# B&R Automation Studio project x20ost (part 6)

#### bnrmessage.h
```c
/********************************************************************
 * COPYRIGHT -- Kontora
 ********************************************************************
 * Program: bnrmain
 * File: bnraninput.h
 * Author: Abramenya
 * Created: January 19, 2009
 *******************************************************************/

#ifndef __MESSAGE_H__
#define __MESSAGE_H__
#include "typedefs.h"
typedef void (*CCPFN)(void);
//Message For My System
#ifdef WIN32
typedef struct _tagCANnode_typ
{
	BOOL enable;
	UINT node_nr;
	UINT status;
}CANnode_typ;

typedef struct _tagCANopen_typ
{
	BOOL enable;
	UINT baud_rate;
	UINT cob_anz;
	UINT device;
}CANopen_typ;

typedef struct _tagFRM_xopen_typ
{
	BOOL   enable;
	UDINT	device;
	UDINT	mode;
	UDINT	config;
	UINT	status;
	UDINT	*ident;
	BYTE	internal[27];
}FRM_xopen_typ;
typedef struct _tagFRM_close_typ
{
	BOOL   enable;
	UDINT  *ident;
	UINT   status;
	BYTE   internal[27];
}FRM_close_typ;
typedef struct _tagXOPENCONFIG
{
	UINT   idle;
	UINT   delimc;
	USINT  delim[2];
	UINT   tx_cnt;
	UINT   rx_cnt;
	UINT   tx_len;
	UINT   rx_len;
	UINT   argc;
	UDINT  *argv;
}XOPENCONFIG;
typedef struct _tagFRM_gbuf_typ
{
	BOOL   enable;
	UDINT  *ident;
	UINT   status;
	UDINT  *buffer;
	UINT	buflng;
	BYTE	internal[27];
}FRM_gbuf_typ;
//Client
typedef struct _tagFRM_rbuf_typ
{
	BOOL   enable;
	UDINT	*ident;
	UDINT	*buffer;
	UINT	buflng;
	UINT	status;
	BYTE	internal[27];
}FRM_rbuf_typ;
typedef struct _tagFRM_robuf_typ
{
	BOOL   enable;
	UDINT	*ident;
	UDINT	*buffer;
	UINT	buflng;
	UINT	status;
	BYTE	internal[27];
}FRM_robuf_typ;
typedef struct _tagFRM_write_typ
{
	BOOL   enable;
	UDINT  *ident;
	UDINT  *buffer;
	UINT   buflng;
	UINT   status;
	BYTE   internal[27];

}FRM_write_typ;
typedef struct _tagFRM_read_typ
{
	BOOL   enable;
	UDINT  *ident;
	UINT   status;
	UDINT  *buffer;
	UINT   buflng;
	BYTE   internal[27];
}FRM_read_typ;
typedef struct _tagSysInfo
{
    BYTE byInfo;
}SYSxinfo_typ;
typedef struct _tagRTCtime_typ
{
    WORD year;
    BYTE month;
    BYTE day;
    BYTE hour;
    BYTE minute;
    BYTE second;
    WORD millisec;
}RTCtime_typ;
int SYSxinfo(SYSxinfo_typ*);
#endif
typedef struct _tagGetParam
{
    WORD wParam0;
	WORD wParam1;
	WORD wParam2;
	WORD wParam3;
}SGETPARAM;
typedef struct _msgPLCCommand
{
    WORD m_swLen;
	BYTE m_sbyFor;
	BYTE m_sbyType;
    BYTE m_sbyDevID;
	BYTE m_sbyInfo[70];
}SPLCCOMM;
typedef struct _msgSystem0
{
    WORD m_swLen;
    BYTE m_sbyFrom;
	BYTE m_sbyFor;
	BYTE m_sbyIntType;
	BYTE m_sbyServerID;
	BYTE m_sbyType;
    BYTE m_sbyDirection;
    BYTE m_sbySensor;
	BYTE m_sbyInfo[350];
}SMESSAGE;
typedef struct _msgSystem00
{
    WORD m_swLen;
    BYTE m_sbyFrom;
	BYTE m_sbyFor;
	BYTE m_sbyIntType;
	BYTE m_sbyServerID;
	BYTE m_sbyType;
    BYTE m_sbyDirection;
    BYTE m_sbySensor;
	BYTE m_sbyInfo[2000];
}SLMESSAGE;
typedef struct _msgShSystem0
{
    WORD m_swLen;
    BYTE m_sbyFrom;
	BYTE m_sbyFor;
	BYTE m_sbyIntType;
	BYTE m_sbyServerID;
	BYTE m_sbyType;
    BYTE m_sbyDirection;
    BYTE m_sbySensor;
	BYTE m_sbyInfo[200];
}SHMESSAGE;
typedef struct _msgShSystem1
{
    WORD m_swLen;
    BYTE m_sbyFrom;
	BYTE m_sbyFor;
	BYTE m_sbyIntType;
	BYTE m_sbyServerID;
	BYTE m_sbyType;
    BYTE m_sbyDirection;
    BYTE m_sbySensor;
	BYTE m_sbyInfo[30];
}SHORTMESSAGE;
typedef struct _tagJob
{
	CCPFN pfnProcAddres;
	BYTE  byPeriod;
	BYTE  byStateProc;
	SINT  chProcName[50];
}SJOBINFO;

typedef struct _tagTcpAddres
{
    BYTE byAddr0;
	BYTE byAddr1;
	BYTE byAddr2;
	BYTE byAddr3;
}STCPADDR;
typedef struct _tagArmInterface
{
	BYTE byNumber;
    BYTE byType;
	BYTE byPortRate;
	BYTE byAmTCPPort;
	DWORD dwpPortNumber[DEV_MAX_TCP_PORT];
	STCPADDR stTcpAddr;
	SINT chTcpAddr[30];
}SARMINTERFACE;
typedef struct _tagHardPinConfig
{
	BYTE byPinNumber;
	BYTE byPinType;
	BYTE byPinState;
	PVOID pvValue;
}SHARDPIN;
typedef struct _tagHardSlotConfig
{
	BYTE bySlotNumber;
	BYTE bySlotType;
	BYTE byPinAmout;
	BYTE byState;
	BYTE byAlmState;
	PVOID pvAlmState;
	PVOID *pvAlmPin;
	PVOID *pvPin;
}SHARDSLOT;
typedef struct _tagKpParam
{
    BYTE byKpID;
	BYTE byStoreMode;
	BYTE byAmCall;
	BYTE byCallPeriod;
	//BYTE bySetChann;
	SINT byPassword[20];
	SINT byPhone0[20];
	SINT byPhone1[20];
	SINT byPhone2[20];
}SKPPARAM;
typedef struct _tagHardComputer
{
    BYTE byComputerType;
	BYTE bySystemID;
    SINT chComputerName[DEV_MAX_TEXT_NAME];
	SINT chProgrammVersion[DEV_MAX_TEXT_NAME];
    SINT chDateOfWrite[DEV_MAX_TEXT_NAME];
	BYTE bySlotAmout;
	BYTE byArmAmout;
	SKPPARAM *pKpParam;
	SARMINTERFACE *pArmInterface[DEV_MAX_ARM_PORT];
	SHARDSLOT sSlot[DEV_MAX_SLOTS_PS260];
}SHARDCOMPUTERTABLE;
typedef struct _tagSensorInitTable
{
    INT  iLoLimitValue;
	INT  iHiLimitValue;
}SENSORINITTABLE;
/*
pT->m_sSNSParam.dY_max    = 20.0;
pT->m_sSNSParam.Kp        = 0.4;
pT->m_sSNSParam.Tn        = 6000.0;
pT->m_sSNSParam.Tv        = 0.0;
pT->m_sSNSParam.Tf        = 1.0;
pT->m_sSNSParam.Kw        = 1.0;
pT->m_sSNSParam.Kfbk      = 1.0;
pT->m_sLCPid.A            = 0;//500;
pT->m_sLCPid.Y_man	      = 0;
*/
typedef struct _tagSensorParamTable
{
    REAL m_swResistance;
    REAL m_swHiLimit;
    REAL m_swLoLimit;
    REAL m_swHiAlLimit;
    REAL m_swLoAlLimit;
    REAL m_swHiOper;
    REAL m_swLoOper;
    REAL m_swInitValue;
	REAL m_rlDy;
	REAL m_rlKp;
	REAL m_rlTn;
	REAL m_rlKw;
	REAL m_rlKfbk;
	REAL m_rlTv;
	REAL m_rlTf;
	INT16 m_rlA;
	INT16 m_rlYman;
	BYTE m_byFilterOn;
	BYTE m_swPidDiffMode;
	WORD m_swMaxAcpInp;
	WORD m_swMaxAcpOut;
	BYTE m_byID;
    BYTE bySrcSlotNumber;
	BYTE bySrcPinNumber;
    BYTE m_snType;
    BYTE m_sbyParamType;
    BYTE m_sbyInpState;
    BYTE m_sbyOutState;
    BYTE m_sbyMode;
	BYTE m_sbyPmode;
	BYTE m_sbyOmode;
	REAL m_srOmin;
	REAL m_srOmax;
	WORD m_swOpenTime;
	SINT m_chSNname[10];
}SNSPARAMTABLE;

typedef struct _tagOutGate
{
	WORD wLoLimit;
	WORD wHiLimit;
	WORD wCurrOpen;
	WORD wOpenTime;
	REAL rMinRamp;
	REAL rMaxRamp;
	BYTE byOType;
	BYTE byMode;
	BYTE byID;
	BYTE byType;
    BYTE byOutSlotNumber;
	BYTE byOutPinNumber;
	SINT chName[10];
}SOUTGATE;
typedef struct _tagSensorInputGates
{
  BYTE byAmInGate;
  SNSPARAMTABLE mIn[12];
}SINPUTGATE;
typedef struct _tagSensorOutputGates
{
	BYTE byAmOutGate;
	SOUTGATE mOut[12];
}SOUTPUTGATE;
typedef struct _tagPinGate
{
	BYTE sbySlot;
	BYTE sbyPin;
}SPINGATE;
typedef struct _tagDigitalGate
{
    WORD swAmpin;
	SPINGATE sPinGate[32];
}SDIGGATE;
typedef struct _tagDigitalGates
{
    BYTE byAmGate;
	SDIGGATE sIoGate[10];
}SDIGGATES;
typedef struct _tagSwitchingTable
{
    #if MYSYSTEM_ID != 5
	 BYTE bySensorID;
	 PVOID sSensorParamTable;
	 TStateList *m_pStateList;
	 BYTE bySwitchCommand;
	 BOOL blEnable;
	 BYTE byAmOutGate;
	 PVOID sOutGate[DEV_AMT_GATE_SNS];
	#else
	 BYTE bySensorID;
     BYTE bySlot;
	 BYTE byPin;
	 BYTE byType;
    #endif
}SSWITCHTABLE;
typedef struct _tagDirectionTable
{
    BYTE byDirectionID;
	BYTE byDirectionCode;
	BYTE byAmSwitching;
	BYTE byAmTI;
	BYTE byAmTS;
	BYTE byAmTU;
	BYTE byAmTR;

	PVOID pvIn;
	PVOID pvOut;
	PVOID pSwitchTable[DEV_AMT_SWC_IDIR];
}SDIRTABLE;
typedef struct _tagSoftSwitchingConfig
{
	BYTE byTableVersion;
	SINT chTableVersionName[DEV_MAX_TEXT_NAME];
	BYTE byAmDirection;
	SDIRTABLE sDirectionTable[DEV_AMT_DIR_INST];
}SSOFTSWITCHTABLE;
//Kp Tag
typedef struct _tagTime
{
    BYTE tDay;
	BYTE tMonth;
	BYTE tYear;
	BYTE tHour;
	BYTE tMin;
	BYTE tSec;
	BYTE tMSecL;
	BYTE tMSecH;
}STIME;
typedef struct _tagKpEvent
{
	WORD wLen;
	BYTE byType;
    BYTE byAddr;
	BYTE byCause;
    WORD wValue;
    STIME sTime;
}SKPEVENT;
typedef struct _tagQueryReqAddr
{
	WORD wSize;
	BYTE byA0;
	BYTE byA1;
	BYTE byA2;
}SREGADDR;
typedef struct _tagReqParam
{
	WORD wSize;
	WORD wParam;
	BYTE byA0;
	BYTE byA1;
	BYTE byA2;
}SREGPARAM;
//Датчик температуры
typedef struct _tagTTMData
{
	WORD wJob;
	WORD wParam;
}STTMDATA;
/*
typedef struct _tagTTMDatas
{
	BYTE Count;
	BYTE byType;
	STTMDATA sDT[2];
}STTMDATAS;
*/
typedef struct _tagTTMParam
{
	BYTE byID;
	BYTE byAmParam;
	BYTE byType;
	BYTE bySlot;
	BYTE byPin;
	BYTE byAlmState;
	BYTE byState;
	STTMDATA sDT;
}STTMPARAM;
typedef struct _tagTTMParams
{
	BYTE byAmSlot;
	BYTE byType;
	STTMPARAM sTTM[4];
}STTMPARAMS;
//Датчик давления
typedef struct _tagTPRData
{
	WORD wJob;
	WORD wParam;
}SPRMDATA;
/*
typedef struct _tagTPRDatas
{
	BYTE Count;
	BYTE byType;
	SPRMDATA sDT[2];
}SPRMDATAS;
*/
typedef struct _tagTPRParam
{
	BYTE byID;
	BYTE byAmParam;
	BYTE byType;
	BYTE bySlot;
	BYTE byPin;
	BYTE byAlmState;
	BYTE byState;
	SPRMDATA sDT;
}STPRPARAM;
typedef struct _tagTPRParams
{
	BYTE byAmSlot;
	BYTE byType;
	STPRPARAM sTPR[4];
}STPRPARAMS;
//Счетчики
typedef struct _tagTCData
{
	REAL fKoeff;
	DWORD dwParam;
}STCDATA;
/*
typedef struct _tagTCDatas
{
	BYTE Count;
	BYTE byType;
	STCDATA sDT[16];
}STCDATAS;
*/
typedef struct _tagTCParam
{
	BYTE byID;
	BYTE byAmParam;
	BYTE byType;
	BYTE bySlot;
	BYTE byPin;
	BYTE byAlmState;
	BYTE byState;
	DWORD dwMaxFreq;
	STCDATA sDT;
}STCPARAM;
typedef struct _tagTCParams
{
	BYTE byAmSlot;
	BYTE byType;
	STCPARAM sTC[18];
}STCPARAMS;
//Управляемые краны
typedef struct _tagTKData
{
	BYTE byStOP;
	BYTE byStCL;
	BYTE byStMD;
    WORD wMaxOpenTime;
    REAL fJobOpen;
    REAL fOpenState;
}STKDATA;
/*
typedef struct _tagTKDatas
{
	BYTE Count;
	BYTE byType;
	STKDATA sDT[4];
}STKDATAS;
*/
typedef struct _tagTKParam
{
	BYTE byID;
	BYTE byAmParam;
	BYTE byType;
	BYTE bySlot;
	BYTE byPin;
	BYTE bySlot1;
	BYTE byPin1;
    STKDATA sDT;
}STKPARAM;
typedef struct _tagTKParams
{
	BYTE byAmSlot;
	BYTE byType;
	STKPARAM sTK[5];
}STKPARAMS;
//Измеритель уровня
typedef struct _tagLVData
{
	WORD wSt0;
	WORD wJob0;
	WORD wJob1;
	WORD wParam;
}SLVDATA;
/*
typedef struct _tagPUDatas
{
	BYTE Count;
	BYTE byType;
	SPUDATA sDT[2];
}SPUDATAS;
*/
typedef struct _tagLVParam
{
	BYTE byID;
	BYTE byAmParam;
	BYTE byType;
	BYTE bySlot;
	BYTE byPin;
	BYTE bySlot1;
	BYTE byPin1;
    SLVDATA sDT;
}SLVPARAM;
typedef struct _tagLVParams
{
	BYTE byAmSlot;
	BYTE byType;
	SLVPARAM sLV[2];
}SLVPARAMS;
//Переключатель режима
typedef struct _tagPLData
{
	BYTE byParam;
}SPLDATA;
typedef struct _tagPLParam
{
	BYTE byID;
	BYTE byAmParam;
	BYTE byType;
	BYTE bySlot;
	BYTE byPin;
    SPLDATA sDT;
}SPLPARAM;
typedef struct _tagPLParams
{
	BYTE byAmSlot;
	BYTE byType;
	SPLPARAM sPL[2];
}SPLPARAMS;
//Таймер операции
typedef struct _tagTMData
{
	WORD wJob;
	WORD wParam;
}STMDATA;
typedef struct _tagTMParam
{
	BYTE byID;
	BYTE byAmParam;
	BYTE byType;
	BYTE bySlot;
	BYTE byPin;
    STMDATA sDT;
}STMPARAM;
typedef struct _tagTMParams
{
	BYTE byAmSlot;
	BYTE byType;
	STMPARAM sTM[2];
}STMPARAMS;
//Перекидное устройство
typedef struct _tagPUData
{
	WORD wSt0;
	WORD dwTimeConst;
	WORD dwOpenTime;
}SPUDATA;
/*
typedef struct _tagPUDatas
{
	BYTE Count;
	BYTE byType;
	SPUDATA sDT[2];
}SPUDATAS;
*/
typedef struct _tagPUParam
{
	BYTE byID;
	BYTE byAmParam;
	BYTE byType;
	BYTE bySlot;
	BYTE byPin;
	BYTE bySlot1;
	BYTE byPin1;
	BYTE bySlot2;
	BYTE byPin2;
	BYTE bySlot3;
	BYTE byPin3;
    SPUDATA sDT;
}SPUPARAM;
typedef struct _tagPUParams
{
	BYTE byAmSlot;
	BYTE byType;
	SPUPARAM sTPU[2];
}SPUPARAMS;
//Частотный привод
typedef struct _tagTFData
{
	//BYTE byStartST;
	//BYTE byStopST;
	//BYTE byAlST0;
	//BYTE byAlST1;
    WORD wSt0;
	WORD wTask;
	WORD wParam;
}STFDATA;
/*
typedef struct _tagTFDatas
{
	BYTE Count;
	BYTE byType;
	STFDATA sDT[3];
}STFDATAS;
*/
typedef struct _tagTFParam
{
	BYTE byID;
	BYTE byAmParam;
	BYTE byType;
	BYTE bySlot; //Для задания
	BYTE byPin;  //Для задания

	BYTE bySlot1; //Запуск
	BYTE byPin1;  //Запуск

	BYTE bySlot2; //Останов
	BYTE byPin2;  //Останов

	BYTE bySlot3; //Авария1
	BYTE byPin3;  //Авария1

	BYTE bySlot4; //Авария2
	BYTE byPin4;  //Авария2
    STFDATA sDT;
}STFPARAM;
typedef struct _tagTFParams
{
	BYTE byAmSlot;
	BYTE byType;
	STFPARAM sTF[4];
}STFPARAMS;
//Телеиндикация
typedef struct _tagTIParam
{
	BYTE byID;
	BYTE byAmParam;
	BYTE byType;
	BYTE bySlot;
	BYTE byPin;
	BYTE byAlmState;
	BYTE byState;
	BYTE byPriority;
	BYTE byDrTimer;
	WORD wHiLimit;
	WORD wHiGister;
	WORD wLoGister;
	WORD wLoLimit;
	WORD wLo;
	WORD wHi;
	WORD wEvPercent;
	WORD wParam;
}STIPARAM;
typedef struct _tagTIParams
{
	BYTE byAmSlot;
	BYTE byType;
	STIPARAM sTI[32];
}STIPARAMS;

//Весы
typedef struct _tagTVSData
{
	BYTE byData[11];
}STVSDATA;
typedef struct _tagTVSParam
{
	BYTE byID;
	BYTE byAmParam;
	BYTE byType;
	STVSDATA sDT;
}STVSPARAM;
typedef struct _tagTVSarams
{
	BYTE byAmSlot;
	BYTE byType;
	STIPARAM sTVS[2];
}STVSPARAMS;
//Телесигнализация(дискретное)
typedef struct _tagTSParam
{
	BYTE byID;
	BYTE byAmParam;
	BYTE byType;
	BYTE bySlot;
	BYTE byPin;
	BYTE byAlmState;
	BYTE byState;
	BYTE byPriority;
	BYTE byCRemPulce;
    BYTE byCSetPulce;
	BYTE byAlarmMode;
    BYTE byParam;
}STSPARAM;
typedef struct _tagTSParams
{
	BYTE byAmSlot;
	BYTE byType;
	STSPARAM sTS[20];
}STSPARAMS;

//Телесигнализация1(дискретное)
typedef struct _tagTSMData
{
	BYTE byParam;
}STSMDATA;
/*
typedef struct _tagTSMDatas
{
	BYTE Count;
	BYTE byType;
	STSMDATA sDT[19];
}STSMDATAS;
*/
typedef struct _tagTSMParam
{
	BYTE byID;
	BYTE byAmParam;
	BYTE byType;
	BYTE bySlot;
	BYTE byPin;
	BYTE byAlmState;
	BYTE byState;
	BYTE byPriority;
	BYTE byCRemPulce;
    BYTE byCSetPulce;
	BYTE byAlarmMode;
    STSMDATA sDT;
}STSMPARAM;
typedef struct _tagTSMParams
{
	BYTE byAmSlot;
	BYTE byType;
	STSPARAM sTS[20];
}STSMPARAMS;

//Аварии
typedef struct _tagTALData
{
	WORD wParam;
}STALDATA;
typedef struct _tagTALaram
{
	BYTE byID;
	BYTE byAmParam;
	BYTE byType;
	BYTE bySlot;
	BYTE byPin;
	BYTE byAlmState;
	BYTE byState;
    STALDATA sDT;
}STALPARAM;
typedef struct _tagTALParams
{
	BYTE byAmSlot;
	BYTE byType;
	STALPARAM sTA[2];
}STALPARAMS;

//Телеуправление(дискретное)
typedef struct _tagTUParam
{
	BYTE byID;
	BYTE byAmParam;
	BYTE byType;
	BYTE bySlot;
	BYTE byPin;
	BYTE byAlmState;
	BYTE byState;
	BYTE byPulceType;
    BYTE byCSetPulce;
	BYTE byParam;
}STUPARAM;
typedef struct _tagTUParams
{
	BYTE byAmSlot;
	BYTE byType;
	STUPARAM sTU[64];
}STUPARAMS;

//Телеуправление1(дискретное)
typedef struct _tagTUMData
{
	BYTE byParam;
}STUMDATA;
typedef struct _tagTUMParam
{
	BYTE byID;
	BYTE byAmParam;
	BYTE byType;
	BYTE bySlot;
	BYTE byPin;
	BYTE byAlmState;
	BYTE byState;
	BYTE byPulceType;
    DWORD byCSetPulce;
	STUMDATA sDT;
}STUMPARAM;
typedef struct _tagTUMParams
{
	BYTE byAmSlot;
	BYTE byType;
	STUMPARAM sTU[16];
}STUMPARAMS;

//Модуль слежения
typedef struct _tagODSData
{
	//BYTE byAutoStart;
	//BYTE byPreStart;
	//BYTE byStart;
	//BYTE byStop;
	//BYTE byFinish;
    //BYTE byMode;
    DWORD wSt0;
	WORD wJTMPreStart;
	WORD wTMPreStart;
	WORD wJTMStart;
	WORD wTMStart;
	WORD wJTMWait;
	WORD wTMWait;
}SOBSMDATA;
typedef struct _tagOBSParam
{
	BYTE byID;
	BYTE byAmParam;
	BYTE byType;
	BYTE bySlot;
	BYTE byPin;
	BYTE byAlmState;
	BYTE byState;
	SOBSMDATA sDT;
}SOBSPARAM;
typedef struct _tagOBSParams
{
	BYTE byAmSlot;
	BYTE byType;
	SOBSPARAM sOS[1];
}SOBSPARAMS;

/*
&nTPR,
&nTTM,
&nTC,
&nTF,
&nTKP,
&nTPU,
&nTS,
&nTU,
*/
typedef struct _tagObserveTable
{
    SPRMDATA nTPR[2];
    STTMDATA nTTM[2];
	STCDATA  nTC[16];
	STFDATA  nTF[3];
	STKDATA  nTKP[4];
	SPUDATA  nPU[2];
	STSMDATA nTS[15];
	STUMDATA nTU[10];
	STVSDATA nTVS[2];
	SLVDATA  nLV[1];
	SPLDATA  nPL[1];
	STMDATA  nTM[1];
	STALDATA nTAL[2];
}STOUTTBL;
typedef struct _tagCDataCommand
{
     WORD wDeviceID;
     BYTE byParam0;
     BYTE byParam1;
     BYTE byParam2;
     WORD wParam0;
     WORD wParam1;
     WORD wParam2;
     REAL fParam0;
     REAL fParam1;
     REAL fParam2;
}CDataCommand;
typedef struct _tagContenstTable
{
	BYTE byKpID;
	BYTE byDefSett;
	//#if (MYSYSTEM_ID == 0)||(MYSYSTEM_ID == 1)||(MYSYSTEM_ID == 2)||(MYSYSTEM_ID == 3)
	//REAL mInResistance[16];
    //SINPUTGATE  sInGate;
    ///SOUTPUTGATE sOutGate;
	//WORD m_wLayerMode;
    //#elif MYSYSTEM_ID == 4
	//DWORD m_dwOutState[32];
    //#elif MYSYSTEM_ID == 5
	SKPPARAM  sKP;
	SARMINTERFACE sARM;
	STIPARAMS sTI;
	STSPARAMS sTS;
	STUPARAMS sTU;
    //#endif
}SCONTENSTTABLE;
#endif
```

#### bnrmodule101.h
```c
/********************************************************************
 * COPYRIGHT -- Kontora
 ********************************************************************
 * Program: bnrmain
 * File: bnraninput.h
 * Author: Abramenya
 * Created: January 19, 2009
 *******************************************************************/

#ifndef __MODULE101_H__
#define __MODULE101_H__
#include "typedefs.h"
#include "bnrcyclicsystem.h"
#include "bnrregedit.h"
Class CModule101
{
	 void (*CCModule101)(This);
	 void (*DCModule101)(This);
Public
     void (*Init)(This);
     BOOL (*LoLevelHandler)(This,SMESSAGE *pMsg);
     BOOL (*HiLevelHandler)(This,SMESSAGE *pMsg);
	 BOOL (*SendMessage)(This,BYTE,BYTE);
	 BYTE (*CreateCRC)(This,BYTE *pMsg,BYTE byLen);
	 BYTE (*AddADSU)(This,BYTE *pMsg,BYTE byNum);
	 BYTE (*AddADSU1)(This,BYTE *pMsg,BYTE byNum);
	 BYTE (*PackADSU)(This,BYTE *pMsg);
	 WORD (*GetW)(This,BYTE *pbyParam);
	 BOOL (*GetSettings)(This);
	 BOOL (*SetSettings)(This);
	 void (*CopyW)(This,PVOID pvDst,PVOID pvSrc);
	 BOOL (*SendBroadcast)(This,SMESSAGE *pMsg);
	 BYTE (*AddBroadADSU)(This,BYTE *pMsg,SKPEVENT *pEV);
	 BOOL (*Autorisation)(This,WORD wKeyCode,BYTE byKpID);
     Virtual BOOL (*HandleTask)(This,TTask* pvTask);
     Virtual BOOL (*EventHandler)(This,SMESSAGE *pMsg);
	 Virtual TStateList* (*GetStateList)(This);
     //Virtual void (*CyclicProc)(This);
	 DECLARE_IMPLEMENT_BASE(CCyclicSystem)
Private
     CRegModule m_nRM;
     BYTE m_byModuleID;
	 BOOL m_blRepFree;
	 //STISTAG  m_sTiTsMsg;
	 SREGADDR m_pA;
	 SREGPARAM m_nRD;
	 SMESSAGE *m_pOutMsg;
	 SMESSAGE m_sOutMsg;
	 SMESSAGE m_sSvOutMsg;
}
DECLARE_DEFINITION(CModule101)
#define TIMER_SRR_00 10

/*
typedef struct   {
BYTE bt0; // аҐ§Ґаў ў ­ з «Ґ
BYTE bt1; //
BYTE Len;
unsigned nGlUnit:6; //ЙНННН»
unsigned nLocUnit:5;//є    є
unsigned nP1:4;      //є ID є
unsigned bit1:1;
unsigned nP2:11;
unsigned nP3:5;
BYTE Data[0x100-7];
} MSG_FPO1;
*/
typedef struct _tagAdsuHead
{
    BYTE Type;
    BYTE VSQ;
    BYTE Cause;
    //BYTE Ordinator;
    BYTE CAA00;
    BYTE CAA01;
}SADSUHEAD;
typedef struct _tagIEA
{
    BYTE IOA00;
    BYTE IOA01;
    BYTE IOA02;
}SIEA;
typedef struct _tagSIQ
{
	BYTE SPI:1;
	BYTE RES:3;
	BYTE BL:1;
	BYTE SB:1;
	BYTE NT:1;
	BYTE IV:1;
}SIQ;
typedef struct _tagTime24
{
    BYTE MSecL;
	BYTE MSecH;
	BYTE Min:6;
	BYTE Res:1;
	BYTE IV:1;
}STIME24;
typedef struct _tagNVA
{
    BYTE byNvaL;
	BYTE byNvaH;
}NVA;
typedef struct _tagFDCO
{
    BYTE IOA00;
    BYTE IOA01;
    BYTE IOA02;
	BYTE DCS:4;
	BYTE BL:1;
	BYTE SB:1;
	BYTE NT:1;
	BYTE IV:1;
    BYTE MSecL;
	BYTE MSecH;
	BYTE Min:6;
	BYTE Rest:1;
	BYTE IVt:1;
}FDCO;

typedef struct _tagFTIME
{
    BYTE IOA00;
    BYTE IOA01;
    BYTE IOA02;
	BYTE MSecL;
	BYTE MSecH;
	//BYTE IV:1;
	//BYTE Res1:1;
	BYTE Min;

	//BYTE SU:1;
	//BYTE Res2:2;
	BYTE Hour;

	//BYTE DayN:3;
	BYTE DayM;

	//BYTE Res3:4;
	BYTE Month;

	//BYTE Res4:1;
	BYTE Year;
}FTIME;

typedef struct _tagFSIQ
{
    BYTE IOA00;
    BYTE IOA01;
    BYTE IOA02;

	BYTE SPI:1;
	BYTE RES:3;
	BYTE BL:1;
	BYTE SB:1;
	BYTE NT:1;
	BYTE IV:1;
    BYTE MSecL;
	BYTE MSecH;
	BYTE Min:6;
	BYTE Rest:1;
	BYTE IVt:1;
}FSIQ;
typedef struct _tagFNVA
{
    BYTE IOA00;
    BYTE IOA01;
    BYTE IOA02;
    BYTE byNvaL;
	BYTE byNvaH;
	BYTE OV:1;
	BYTE RES:3;
	BYTE BL:1;
	BYTE SB:1;
	BYTE NT:1;
	BYTE IV:1;
}FNVA;
typedef struct _tagFTNVA
{
    BYTE IOA00;
    BYTE IOA01;
    BYTE IOA02;
    BYTE byNvaL;
	BYTE byNvaH;

	BYTE byQDS;
    /*#ifdef WIN32
    BYTE MSecL;
	BYTE MSecH;
	BYTE Min:6;
	BYTE Res1:1;
	BYTE IV:1;
	BYTE Hour:5;
	BYTE Res2:2;
	BYTE SU:1;
	BYTE DayM:5;
	BYTE DayN:3;
	BYTE Month:4;
	BYTE Res3:4;
	BYTE Year:7;
	BYTE Res4:1;
	#else
	*/
    BYTE MSecL;
	BYTE MSecH;
	BYTE Min;
	BYTE Hour;
	BYTE DayM;
	BYTE Month;
	BYTE Year;

	/*
	BYTE IV:1;
	BYTE Res1:1;
	BYTE Min:6;

	BYTE SU:1;
	BYTE Res2:2;
	BYTE Hour:5;

	BYTE DayN:3;
	BYTE DayM:5;

	BYTE Res3:4;
	BYTE Month:4;

	BYTE Res4:1;
	BYTE Year:7;
	*/
	//#endif
}FTNVA;
enum _tagAuto101Value
{
	 FCB=0,
	 FCV,
	 ACD,
	 DFC,
	 MFCB,
	 MFCV,
     CACK,
	 MCMD,
	 ISERROR,
	 ISCHNG,
	 ISCHNGTI,
	 ONE,
	 ZERO,
	 VAL0,
	 STATE_101,
	 STATE_WSY,
};
enum
{
	TMR_SRR=0,
	TMR_SSC,
};
#endif
```

#### bnrmysystem.h
```c
/********************************************************************
 * COPYRIGHT -- Kontora
 ********************************************************************
 * Program: bnrmain
 * File: bnraninput.h
 * Author: Abramenya
 * Created: January 19, 2009
 *******************************************************************/

#ifndef __MYSYSTEM_H__
#define __MYSYSTEM_H__
#include "typedefs.h"
#include "bnrmessage.h"
#include "bnrprocmanager.h"
#include "bnradmin.h"
#include "bnrcomputer.h"
#include "bnrobserve.h"
#include "bnrpob.h"
#include "bnrkp.h"
#include "bnrmodule101.h"
#include "bnrcomserver.h"
#include "bnrtcpserver.h"
#include "bnrcomvs0.h"
#include "bnrcomvs1.h"
#include "bnrtcpserver.h"
#include "bnrmeasur.h"
#ifdef WIN32
#include "winsock.h"
void CreateGetProc(PVOID pVoid);
#endif
Class CSystem
{
	 void (*CCSystem)(This);
	 void (*DCSystem)(This);
Public
	 void (*CreateSystem)(This,SHARDCOMPUTERTABLE *pTable);
     void (*CreateAdmin)(This);
     void (*CreateComputer)(This,SHARDCOMPUTERTABLE *pTable);
	 void (*CreateSysBox)(This);
	 void (*CreateObserveModule)(This,SHARDCOMPUTERTABLE *pTable,SSOFTSWITCHTABLE *pSoftSwitchTable);
	 void (*CreateProc)(This);
	 void (*SwitchSystem)(This,SSOFTSWITCHTABLE *pSoftSwitchTable);
	 BOOL (*SendMessage)(This,BYTE byFor,BYTE byType);
	 void (*SendMsg)(This,SMESSAGE*);
 	 Virtual BOOL (*EventHandler)(This,SMESSAGE *pMsg);
	 //Virtual void (*CyclicProc)(This);
Private
     CAdmin *m_pAdmin;
     CComputer *m_pComputer;
     #if MYSYSTEM_ID != 5
	 CObserveModule *m_pObsModule;
     #else
	 CKpModule  *m_pObsModule;
	 #endif
	 CModule101 *m_p101;
	 CComServer *m_nCom;
	 CComVS0    *m_nCVS0;
	 CComVS1    *m_nCVS1;
	 CTcpServer *m_nTCP;
	 CMsModule  *m_nMS;
	 CMTimer m_pResetTimer;
	 BYTE m_blSystemInitState;
	 BOOL m_byTcpConn;
	 BYTE m_byArmAmout;
	 BYTE m_bySystemID;
	 DECLARE_IMPLEMENT_BASE(CCyclicSystem)
}
DECLARE_DEFINITION(CSystem)
_GLOBAL CSystem *m_pSystem;
#endif
```

#### bnrmytimer.h
```c
/********************************************************************
 * COPYRIGHT -- Kontora
 ********************************************************************
 * Program: bnrmain
 * File: bnraninput.h
 * Author: Abramenya
 * Created: January 19, 2009
 *******************************************************************/

#ifndef __MTIMER_H__
#define __MTIMER_H__
#include "typedefs.h"
#include "bnrsystemtimer.h"
#include "bnrmessage.h"
#include "bnrpob.h"
Class CMTimer
{
	 void (*CCMTimer)(This);
	 void (*DCMTimer)(This);
Public
	 void (*SetTimer)(This,BYTE byFor,BYTE byFrom,BYTE byEvent,BYTE byDir,BYTE bySens,BYTE byBox);
     void (*Restart)(This);
     void (*OnTimer)(This,DWORD);
	 void (*OfTimer)(This);
	 DWORD (*GetTime)(This);
	 Virtual void (*DoAction)(This);
Private
     SHORTMESSAGE sMsg;
     DWORD m_dwSTime;
     BYTE m_byFor;
	 BYTE m_byFrom;
	 BYTE m_byEvent;
	 BYTE m_byDir;
	 BYTE m_bySens;
	 BYTE m_byBox;
	 DECLARE_IMPLEMENT_BASE(CSystemTimer)
}
DECLARE_DEFINITION(CMTimer)
#endif
```

#### bnrobserve.h
```c
/********************************************************************
 * COPYRIGHT -- Kontora
 ********************************************************************
 * Program: bnrmain
 * File: bnraninput.h
 * Author: Abramenya
 * Created: January 19, 2009
 *******************************************************************/
//
#ifndef __DIRMODULE_H__
#define __DIRMODULE_H__
#include "typedefs.h"
#if MYSYSTEM_ID != 5
#include "bnrcyclicsystem.h"
#include "bnrdirmodule.h"
#include "bnrmytimer.h"
#include "bnradmin.h"
#include "bnrflash.h"
typedef void (*PFNVOID)(void);
Class CObserveModule
{
	void (*CCObserveModule)(This);
	void (*DCObserveModule)(This);
Public
	void (*Init)(This,SSOFTSWITCHTABLE *pSoftSwitchTable);
	void (*CreateObserve)(This,SSOFTSWITCHTABLE *pSoftSwitchTable);
	void (*ConnectToComputer)(This,CComputer *pComputer);
	void (*SetSystemID)(This,BYTE);
	void (*GetObserveData)(This,BYTE byEvent);
	CDirectionModule* (*GetDirection)(This,BYTE byDir);
    CSensor* (*GetSensor)(This,CDirectionModule**,BYTE,BYTE);
	void (*ConnectToAdmin)(This,CAdmin*);
	Virtual BOOL (*EventHandler)(This,SMESSAGE *pMsg);
    Virtual void (*CyclicProc)(This);
Private
    CMFlash m_nFlash;
    CAdmin *m_pAdmin;
    CComputer *m_pComputer;
    CMTimer m_pRefrechTmr;
	CDirectionModule **m_pDirectionModule;
	SMESSAGE m_nMsg;
	BYTE m_byObserveProc;
	BYTE m_byObsTime;
	BYTE m_bySystemID;
	BYTE m_byTableVersion;
	SINT m_chTableVersionName[DEV_MAX_TEXT_NAME];
	BYTE m_byAmDirection;
	DECLARE_IMPLEMENT_BASE(CCyclicSystem)
}
DECLARE_DEFINITION(CObserveModule)
#endif
#endif
```

#### bnroutgate.h
```c
/********************************************************************
 * COPYRIGHT -- Kontora
 ********************************************************************
 * Program: bnrmain
 * File: bnraninput.h
 * Author: Abramenya
 * Created: January 19, 2009
 *******************************************************************/

#ifndef __OUTGATE_H__
#define __OUTGATE_H__
#include "typedefs.h"
#if MYSYSTEM_ID != 5
#include "bnrhardpin.h"
Class COutGate
{
	 void (*CCOutGate)(This);
	 void (*DCOutGate)(This);
Public
     void (*Init)(This,BYTE byID,BYTE byType,BYTE byOType,BYTE byMode,REAL rMinRamp,REAL rMaxRamp,CPin *pPin,UINT wLo,UINT wHi,UINT wIni,BYTE byState,WORD wBase,WORD wOTime,SINT *pName);
     void (*OpenGate)(This,REAL rOpenState);
	 void (*OpenGateReq)(This,BYTE);
	 void (*StopGate)(This);
	 void (*SetGate)(This,UINT wValue);
	 void (*SetManGate)(This,UINT wValue);
	 void (*SetDefault)(This);
	 UINT (*GetGate)(This);
	 BYTE (*GetPrcGate)(This);
	 void (*RunGate)(This);
	 void (*SetState)(This,BYTE);
	 void (*SetMinRamp)(This,REAL);
	 void (*SetMaxRamp)(This,REAL);
	 void (*SetHiLimit)(This,WORD wValue);
	 void (*SetOutTime)(This,WORD wValue);
Private
     BYTE m_byGateID;
	 BYTE m_byOType;
	 BYTE m_byMode;
     BYTE m_byType;
	 BYTE m_byState;
	 REAL m_rMinRamp;
     REAL m_rMaxRamp;
	 REAL m_wMaxQt;
	 UINT *m_pwOut;
	 UINT m_wOTime;
	 UINT m_wOut;
	 UINT m_wMinRampValue;
	 UINT m_wMaxRampValue;
	 REAL m_wOperGate;
	 UINT m_wBase;
     UINT m_wLoLimit;
     UINT m_wHiLimit;
	 REAL m_wTickOpen;
	 REAL m_wTickConst;
	 UINT m_wCurrOpenState;
	 UINT m_wIniState;
	 DWORD m_wTick;

	 WORD  m_wQTime;
	 DWORD m_dwTime;
	 BOOL  m_blProccState;
	 CPin  *m_pConnectionPin;
	 SINT  m_chName[30];
	 DECLARE_IMPLEMENT
}
DECLARE_DEFINITION(COutGate)
#endif
#endif
```

#### bnrpin.h
```c
/********************************************************************
 * COPYRIGHT -- Kontora
 ********************************************************************
 * Program: bnrmain
 * File: bnraninput.h
 * Author: Abramenya
 * Created: January 19, 2009
 *******************************************************************/

#ifndef __PIN_H__
#define __PIN_H__
#include "typedefs.h"
#include "bnrmessage.h"
#include "bnrdebug.h"
typedef struct _tagSPin
{
	 UINT iValue;
	 BOOL blValue;
}SPIN;
Class CPin
{
	 void (*CCPin)(This);
	 void (*DCPin)(This);
Public
     void (*Init)(This,SHARDPIN*,SHARDPIN*);
     void (*SetSlot)(This,BYTE bySlot);
	 BYTE (*GetState)(This);
	 Virtual PVOID (*GetAddrPin)(This);
	 Virtual void (*InitPin)(This,PVOID);
     Virtual void (*SetPin)(This,SPIN*);
	 Virtual void (*GetPin)(This,SPIN*);
Private
     BOOL m_blPinON;
     BOOL m_blPinOFF;
     BYTE m_byPinNumber;
	 BYTE m_bySlotNumber;
	 BYTE m_byPinState;
	 PVOID m_pvAlmState;
	 DECLARE_IMPLEMENT
}
DECLARE_DEFINITION(CPin)
#endif
```

#### bnrpob.h
```c
#ifndef __BNRPOB_H__
#define __BNRPOB_H__
#define MAXNAMEBUF 20
#include "typedefs.h"
#include "bnrdebug.h"

//#define  DEF_PUT_BOX
//#define  DEF_GET_BOX
//#define  DEF_INF_BOX
//#define  DEF_CRT_BOX
#define BOX_TRANS_SIZE 256
typedef struct pBufferHiLev
{
     BYTE *pb_mBoxCont;
     WORD w_mBoxWrite;
     WORD w_mBoxRead;
     WORD w_mBoxSize;
     WORD w_mBoxCSize;
     WORD w_mBoxMesCt;
}pBOX;
int  FDEFINE(BYTE b_lNmBox,WORD w_lBoxSize);
int  FPUT(BYTE b_lNmBox,BYTE *pb_lInBox);
int  FGET(BYTE b_lNmBox,BYTE *pb_lInBox);
int  FCHECK(BYTE b_lNmBox);
void FDELETE(BYTE b_lNmBox);
void FFREE(BYTE b_lNmBox);
void FINIT(void);
int  FGET1(BYTE b_lNmBox,BYTE *pb_lInBox);
int  FPUT1(BYTE b_lNmBox,BYTE *pb_lInBox);
int  FCHECKM(BYTE b_lNmBox);
void FSMRB(BYTE b_lNmBox);
int  FFREEM(BYTE b_lNmBox);
#endif
```

#### bnrprocmanager.h
```c
/********************************************************************
 * COPYRIGHT -- Kontora
 ********************************************************************
 * Program: bnrmain
 * File: bnraninput.h
 * Author: Abramenya
 * Created: January 19, 2009
 *******************************************************************/

#ifndef __PROCMANAGER_H__
#define __PROCMANAGER_H__
#include "typedefs.h"
#include "bnrcyclicsystem.h"
#include "bnrsystemtimer.h"
#define PRC_MAN_CH_QUANT  1500
Class CProcManager
{
	 void (*CCProcManager)(This);
	 void (*DCProcManager)(This);
Public
     void (*Init)(This,DWORD dwTicTime,BOOL blStatistic);
     void (*SetTicTime)(This,DWORD);
	 void (*GetTimeStatistic)(This);
     BOOL (*Find)(This,SINT *chName);
	 BOOL (*ConnectProc)(This,CCyclicSystem *pCSystem);
	 BOOL (*ConnectTimer)(This,CSystemTimer *pSTimer);
	 BOOL (*DisconnectTimer)(This,CSystemTimer *pSTimer);
	 void (*DeleteProc)(This,SINT *chName);
	 void (*SuspendThread)(This,SINT *chName);
	 void (*ResumeThread)(This,SINT *chName);
	 void (*SuspendAll)(This);
	 void (*ResumeAll)(This);
	 void (*Run)(This);
	 void (*Start)(This);
	 void (*Stop)(This);
Private
     CCyclicSystem *m_nCyclicSystem[DEV_MAX_CYC_PROC];
     CSystemTimer *m_nSystemTimer[DEV_MAX_SYS_TIMR];
     BYTE m_byCheckQuant;
     BOOL m_blState;
	 BOOL m_blStatistic;
     BYTE m_nMaxProc;
	 BYTE m_nMaxTimer;
	 DWORD m_iProcCounter;
	 DWORD m_dwTicTime;
	 DECLARE_IMPLEMENT
}
DECLARE_DEFINITION(CProcManager)
#endif
```

#### bnrregedit.h
```c
/********************************************************************
 * COPYRIGHT -- Kontora
 ********************************************************************
 * Program: bnrmain
 * File: bnraninput.h
 * Author: Abramenya
 * Created: January 19, 2009
 *******************************************************************/

#ifndef __REGEDIT_H__
#define __REGEDIT_H__
#include "typedefs.h"
#include "bnrmessage.h"
#include "bnrpob.h"
Class CRegModule
{
	 void (*CCRegModule)(This);
	 void (*DCRegModule)(This);
Public
     void (*Init)(This);
     BYTE (*QueryParam)(This,SREGADDR *pA);
	 BYTE (*SaveParam)(This,SREGPARAM *pA);
	 BYTE (*CreateKpParam)(This,SREGADDR *pA);
	 BYTE (*CreatePortParam)(This,SREGADDR *pA);
	 BYTE (*CreateHardParam)(This,SREGADDR *pA);
	 BYTE (*CreateSoftTIParam)(This,SREGADDR *pA);
	 BYTE (*CreateSoftTSParam)(This,SREGADDR *pA);
	 BYTE (*CreateSoftTUParam)(This,SREGADDR *pA);
	 BYTE (*CreateSoftTRParam)(This,SREGADDR *pA);

	 BYTE (*SetKpParam)(This,SREGPARAM *pA);
	 BYTE (*SetPortParam)(This,SREGPARAM *pA);
	 BYTE (*SetHardParam)(This,SREGPARAM *pA);
	 BYTE (*SetSoftTIParam)(This,SREGPARAM *pA);
	 BYTE (*SetSoftTSParam)(This,SREGPARAM *pA);
	 BYTE (*SetSoftTUParam)(This,SREGPARAM *pA);
	 BYTE (*SetSoftTRParam)(This,SREGPARAM *pA);
	 void (*CopyW)(This,PVOID pvDst,PVOID pvSrc);
Private
     SSOFTSWITCHTABLE   *m_pSCT;
     SHARDCOMPUTERTABLE *m_pHCT;
	 DECLARE_IMPLEMENT
}
DECLARE_DEFINITION(CRegModule)
#endif
```

#### bnrsensr.h
```c
/********************************************************************
 * COPYRIGHT -- Kontora
 ********************************************************************
 * Program: bnrmain
 * File: bnrsensr.h
 * Author: Abramenya
 * Created: January 23, 2009
 *******************************************************************/
#ifndef __BSSENSOR_H__
#define __BSSENSOR_H__
#include "typedefs.h"
#if MYSYSTEM_ID != 5
#include "bnrdebug.h"
#include "bnrpin.h"
#include "bnrmessage.h"
#include "bnroutgate.h"
#include "bnrauto.h"
#include "bnrmytimer.h"
#include "bnringate.h"
Class CSensor
{
     void (*CCSensor)(This);
	 void (*DCSensor)(This);
Public
     void (*Init)(This,SSWITCHTABLE*);
     void (*InitDigital)(This,SSWITCHTABLE*);
     void (*SetSensorID)(This,BYTE);
     BYTE (*GetSensorID)(This);
	 void (*SetParType)(This,BYTE);
     BYTE (*GetParType)(This);
     void (*SetDirection)(This,PVOID,BYTE);
	 BYTE (*GetDirection)(This);
	 void (*ObserveProc)(This);
     void (*ConnectFCP)(This,CInputGate*);
	 void (*ConnectOutGate)(This,COutGate*);
	 ///////////////////////////////
     void (*SetLoLimit)(This,UINT);
	 void (*SetHiLimit)(This,UINT);
     void (*SetLoAlLimit)(This,INT16);
	 void (*SetHiAlLimit)(This,INT16);
	 ///////////////////////////////
	 void (*EnableInput)(This,BOOL);
	 void (*EnableProc)(This,BOOL);
	 void (*EnableOutput)(This,BOOL);
     ///////////////////////////////
	 void (*SetLoopMode)(This);
	 void (*SetManMode)(This);
	 void (*SetAutoMode)(This);
     ///////////////////////////////
	 void (*Enable)(This);
	 void (*Disable)(This);
	 void (*SetCallBackProc)(This,PCLB);
	 void (*SetState)(This,DWORD dwState);
	 DWORD (*GetState)(This);
	 void (*SendCommand)(This,BYTE byFor,BYTE byType);
	 SPIN* (*GetInput)(This);
	 SPIN* (*GetOutput)(This);
	 //Statistic
	 void (*AddCaptureData)(This,DINT,DINT,DINT);
	 Virtual void (*CaptureData)(This);
	 void (*StartCaptureProc)(This);
	 void (*StopCaptureProc)(This);
	 INT16**(*GetCaptureBuffer)(This);
	 void (*RestartCaptureProc)(This);
     void (*OpenGate)(This);
	 void (*AddData)(This,DINT);
	 void (*CloseGate)(This);
     void (*GetParamTable)(This,BYTE);
     INT16 (*GetWordParam)(This,BYTE *pbyParam);
	 //Event Handler
	 void (*ConnectPinAddres)(This);
	 void (*SEventHandler)(This,SMESSAGE *pMsg);
	 void (*SetEvent)(This,BOOL*,BOOL*,BYTE);
	 void (*SetAutoEvent)(This,BYTE byEvent);
	 Virtual void (*EventGate)(This,BYTE byEvent);
	 //Utilites
	 REAL (*GetRealParam)(This,BYTE *pbyParam);
	 UINT (*GetInParam)(This,REAL nParam);
     void (*CalcGate)(This);
	 UINT (*AcpToInt)(This,UINT);
	 UINT (*IntToAcp)(This,UINT);
	 REAL (*AcpToReal)(This,UINT nAcpCode);
     UINT (*RealToAcp)(This,REAL nParam);
	 void (*SetOutState)(This,BYTE);
	 void (*SetForAll)(This,BYTE byPType,BYTE byPCode,REAL rParam,UINT nParam);
	 void (*SetLEMode)(This);
	 Virtual void (*IncInput)(This,INT16 wParam);
     Virtual void (*GetParam)(This,BYTE);
	 Virtual void (*SetInput)(This,SPIN*);
	 Virtual void (*SetOutput)(This,BYTE,SPIN*);
	 Virtual BYTE (*CheckLimit)(This);
     Virtual void (*PreProc)(This);
     Virtual void (*Processing)(This);
     Virtual void (*PostProc)(This);
	 Virtual void (*InitSensor)(This,PVOID);
	 Virtual void (*RunAutomat)(This);
	 Virtual void (*EventGen)(This);
	 Virtual void (*EventHandler)(This,SMESSAGE*);
	 Virtual void (*Serialize)(This,BOOL byDir);
	 //Automat
	 void (*SetMsgAuto)(This,SMESSAGE*);
	 Virtual BOOL (*HandleTask)(This,TTask* pvTask);
     Virtual TStateList* (*GetStateList)(This);
Private
     UINT m_nInPin;
     UINT m_nOutPin;
	 CInputGate *m_nInp;
	 WORD m_wSnsMode;
	 BYTE m_byPidMode;
	 BOOL m_blSensorState;
	 BOOL m_blInState;
	 BOOL m_blProcState;
	 BOOL m_blOutState;
     PCLB m_pfnCallBackProc;
     DWORD m_dwState;
	 BYTE m_byEvent;
	 SNSPARAMTABLE *m_pvPT;
     SNSPARAMTABLE m_sPT;
	 UINT m_nAcpOutRamp;
	 UINT m_nAcpMin;
	 UINT m_nAcpMax;
	 UINT m_nIniValue;
	 UINT m_iLoLimit;
	 UINT m_iHiLimit;
	 UINT m_iPLoLimit;
	 UINT m_iPHiLimit;
	 UINT m_iPHiOldLimit;
	 UINT m_iLoAlmLimit;
	 UINT m_iHiAlmLimit;
	 UINT m_iIPLoLimit;
	 UINT m_iIPHiLimit;
	 BYTE m_bySystemID;
	 BYTE m_bySensorID;
     BYTE m_bySensorType;
	 BYTE m_bySwitchCommand;
	 BYTE m_byDirection;
	 BYTE m_byParamType;
	 //Statistic
	 BOOL m_blStatState;
	 WORD m_wStatIndex;
	 BOOL m_blCaptureState;
	 WORD m_wStatQuant;
	 DINT m_pwStatBuff[20];
     //Out Gate
	 BYTE m_byAmOutGate;
     WORD m_wAmInput;
     WORD m_wAmOutput;
	 SOUTGATE m_sGT;
	 COutGate *m_pOutGate[DEV_AMT_GATE_SNS];
	 CPin **m_pINP;
     CPin **m_pOUT;
	 BOOL **m_bINP;
	 BOOL **m_bOUT;
	 UINT **m_nINP;
	 UINT **m_nOUT;
	 DWORD m_dwInState;
     DWORD m_dwOutState;
	 //Proc Alarm Gate Clock
	 BOOL m_blAlmLoLevel;
	 BOOL m_blRAlmLoLevel;
     BOOL m_blAlmHiLevel;
     BOOL m_blRAlmHiLevel;
	 BOOL m_blProcLoLevel;
     BOOL m_blProcHiLevel;
	 PVOID m_pvDirection;
	 //Automat
     TStateList *m_pStateList;
	 CMTimer m_nATmr[4];
	 BYTE m_byAutoState;
	 BYTE V0,V1;
	 DWORD m_dwAutoTime;
	 DECLARE_IMPLEMENT_BASE(CAuto)
}
DECLARE_DEFINITION(CSensor)
#endif
#endif
```

#### bnrslide.h
```c
/********************************************************************
 * COPYRIGHT -- Kontora
 ********************************************************************
 * Program: bnrmain
 * File: bnraninput.h
 * Author: Abramenya
 * Created: January 19, 2009
 *******************************************************************/

#ifndef __DEVICESlot_H__
#define __DEVICESlot_H__
#include "typedefs.h"
#include "bnrmessage.h"
#include "bnrpin.h"
Class CSlot
{
	 void (*CCSlot)(This);
	 void (*DCSlot)(This);
Public
     void (*Init)(This,SHARDSLOT *psvSlot);
     Virtual void (*InitSlot)(This,SHARDSLOT *pSlot);
	 Virtual CPin* (*GetPin)(This,BYTE byNumber);
Private
     BYTE m_bySlotNumber;
     BYTE m_bySlotType;
	 BYTE m_byAmPin;
	 BYTE m_byState;
	 PVOID m_pvAlmState;
	 DECLARE_IMPLEMENT
}
DECLARE_DEFINITION(CSlot)
#endif
```

#### bnrsmartsensor.h
```c
/********************************************************************
 * COPYRIGHT -- Kontora
 ********************************************************************
 * Program: bnrmain
 * File: bnraninput.h
 * Author: Abramenya
 * Created: January 19, 2009
 *******************************************************************/

#ifndef __SMARTSENSOR_H__
#define __SMARTSENSOR_H__
#include "typedefs.h"
#if MYSYSTEM_ID != 5
#include "bnrsensr.h"
#ifndef WIN32
//#include "loopconr.h"
#include "loopcont.h"
#endif
#ifdef WIN32
//fbk_mode
#define LCPID_FBK_MODE_INTERN       0
#define LCPID_FBK_MODE_EXTERN       1
#define LCPID_FBK_MODE_EXT_SELECTOR 2
//d_mode
#define LCPID_D_MODE_X              0
#define LCPID_D_MODE_E              1
//calc_mode
#define LCPID_CALC_MODE_EXACT       0
#define LCPID_CALC_MODE_FAST        1

#define LCPID_OUT_MODE_AUTO            1
#define LCPID_OUT_MODE_CLOSE		   4
#define LCPID_OUT_MODE_CLOSE_JOLTFREE  104
#define LCPID_OUT_MODE_FREEZE          5
#define LCPID_OUT_MODE_FREEZE_JOLTFREE 105
#define LCPID_OUT_MODE_MAN             2
#define LCPID_OUT_MODE_MAN_JOLTFREE    102
#define LCPID_OUT_MODE_OFF             0
#define LCPID_OUT_MODE_OPEN            3
#define LCPID_OUT_MODE_OPEN_JOLTFREE   0

typedef struct _tagSnsParam
{
	 BOOL enable;
     BOOL enter;
     INT16 Y_max;
     INT16 Y_min;
	 REAL dY_max;
     REAL Kp;
	 REAL Tn;
     REAL Tv;
	 REAL Tf;
	 REAL Kw;
     REAL Kfbk;
	 USINT fbk_mode;
     USINT d_mode;
     USINT calc_mode;
     UINT status;
     UDINT *ident;
}LCPIDpara_typ;
typedef struct _tagLcPid
{
	 BOOL enable;
	 UDINT *ident;
	 INT16 W;
	 INT16 X;
	 INT16 A;
	 INT16 Y_man;
	 INT16 Y_fbk;
	 BOOL hold_I;
	 USINT out_mode;
	 UDINT basetime;
	 UINT status;
	 DINT e;
	 INT16 Y;
	 DINT Yp;
	 DINT Yi;
	 DINT Yd;
	 UDINT time_old;
	 DINT Tv_Tf_old;
	 BOOL enable_old;
	 DINT e_old;
}LCPID_typ;
typedef struct _tagCounter
{
	 UDINT muscnt;
	 UDINT mus100cnt;
	 UDINT mscnt;
	 UDINT ms100cnt;
	 UDINT seccnt;
}LCCounter_typ;
typedef struct _tagLcRprt2
{
	 BOOL enable;
	 REAL V;
	 REAL T1;
	 REAL T2;
	 REAL x;
	 REAL y_set;
	 USINT set;
	 REAL y;
	 UINT status;
}LCRPT2_typ;
void LCPIDpara(LCPIDpara_typ *pPara);
void LCPID(LCPID_typ *pPid);
void LCCounter(LCCounter_typ *pCounder);
void LCRPT2(LCRPT2_typ *pLowPas);
#endif
typedef struct _tagPidParam
{
    REAL  Kp;
    REAL  Tn;
    REAL  Tv;
    REAL  Tf;
    REAL  Kw;
    REAL  Kfbk; //24
    REAL  dY_max;
    INT16 Y_max;
    INT16 Y_min;
    INT16 W;
    INT16 X;
    INT16 A;
    INT16 Y_man; //14
	BYTE  enable;
	BYTE  out_mode;
	BYTE  enabled; //3 41
}SPIDPARAM;
Class CSmartSensor
{
	 void (*CCSmartSensor)(This);
	 void (*DCSmartSensor)(This);
	 void (*SetMode)(This,USINT);
	 void (*SetState)(This,BOOL);
	 BOOL (*GetState)(This);
Public
     Virtual void (*InitSensor)(This,PVOID pParam);
     Virtual void (*PreProc)(This);
     Virtual void (*Processing)(This);
     Virtual void (*PostProc)(This);
	 Virtual void (*GetParam)(This,BYTE byOwner);
	 Virtual void (*IncInput)(This,INT16);
	 Virtual void (*SetInput)(This,SPIN*);
	 Virtual void (*SetOutput)(This,BYTE,SPIN*);
	 Virtual void (*EventHandler)(This,SMESSAGE*);
	 Virtual void (*CaptureData)(This);
	 Virtual void (*RunAutomat)(This);
	 Virtual void (*EventGen)(This);
	 Virtual void (*Serialize)(This,BOOL byDir);
	 DWORD (*MotToInt)(This,DWORD dwData);
Private
	 UINT m_wExtError;
     USINT m_byMode;
     BOOL m_blState;
	 INT16 m_iInpV;
     LCPIDpara_typ m_sSNSParam;
     LCPID_typ m_sLCPid;
	 LCCounter_typ m_sCounter;
	 DECLARE_IMPLEMENT_BASE(CSensor)
}
DECLARE_DEFINITION(CSmartSensor)
#endif
#endif
```

#### bnrsystemtimer.h
```c
/********************************************************************
 * COPYRIGHT -- Kontora
 ********************************************************************
 * Program: bnrmain
 * File: bnraninput.h
 * Author: Abramenya
 * Created: January 19, 2009
 *******************************************************************/

#ifndef __SYSTEMTIMER_H__
#define __SYSTEMTIMER_H__
#include "typedefs.h"
Class CSystemTimer
{
	 void (*CCSystemTimer)(This);
	 void (*DCSystemTimer)(This);
	 void (*RunTimer)(This);
	 void (*OnTimer)(This,DWORD);
	 void (*OfTimer)(This);
	 void (*SetTimerID)(This,BYTE);
     Virtual void (*DoAction)(This);
Public
	 DECLARE_IMPLEMENT
     BOOL m_blTimerState;
	 DWORD m_dwTime;
	 BYTE m_byTimerID;
}
DECLARE_DEFINITION(CSystemTimer)
#endif
```

#### bnrtelecontrol.h
```c
/********************************************************************
 * COPYRIGHT -- Kontora
 ********************************************************************
 * Program: bnrmain
 * File: bnraninput.h
 * Author: Abramenya
 * Created: January 19, 2009
 *******************************************************************/

#ifndef __TELECTRL_H__
#define __TELECTRL_H__
#include "typedefs.h"
#include "bnrtelesensor.h"
enum _enTUCommand
{
     EN_STT_PULCE=9,
	 EN_STT_SIGN =10,
};
#define DEF_PULCE 20
Class CTeleControl
{
	 void (*CCTeleControl)(This);
	 void (*DCTeleControl)(This);
Public
     void (*SetPulce)(This);
     Virtual BOOL (*EventHandler)(This,SMESSAGE *pMsg);
     Virtual void (*InitTCHN)(This,PVOID psTable);
     Virtual void (*PreProc)(This);
     Virtual void (*Processing)(This);
	 Virtual void (*PostProc)(This);
	 Virtual void (*SetInPinEvent)(This);
	 Virtual void (*SaveAlarmPin)(This);
	 Virtual void (*SendObsrveMsg)(This);
Public
	 STUPARAM *pP;
     //BOOL m_blSetAlarm;
     BYTE m_bySetPulce;
	 BYTE m_byStPulce;
	 BOOL *m_pbOT;
	 DECLARE_IMPLEMENT_BASE(CTeleSensor)
}
DECLARE_DEFINITION(CTeleControl)
#endif
```

#### bnrteleind.h
```c
/********************************************************************
 * COPYRIGHT -- Kontora
 ********************************************************************
 * Program: bnrmain
 * File: bnraninput.h
 * Author: Abramenya
 * Created: January 19, 2009
 *******************************************************************/

#ifndef __TELEIND_H__
#define __TELEIND_H__
#include "typedefs.h"
#include "bnrtelesensor.h"
enum _tagEnTIParam
{
	 EN_HIL_PR=0,
	 EN_HIG_PR,
	 EN_LOL_PR,
	 EN_LOG_PR,
	 EN_DTM_PR,
};
#define DEF_HILIMIT 29000
#define DEF_HIGISTR 28000
#define DEF_LOLIMIT 19000
#define DEF_LOGISTR 18000
#define DEF_DRTIMER 20
Class CTeleInd
{
	 void (*CCTeleInd)(This);
	 void (*DCTeleInd)(This);
Public
     WORD (*CheckTI)(This);
	 void (*SetEventHi)(This,BOOL *bl0,BOOL *bl1,BYTE byEvent);
	 void (*SetEventTimerHi)(This,BYTE byEvent);
	 void (*SetEventLo)(This,BOOL *bl0,BOOL *bl1,BYTE byEvent);
	 void (*SetEventTimerLo)(This,BYTE byEvent);
	 void (*SetChandgeTimer)(This,BYTE byEvent);
	 void (*InitMeter)(This);
	 void (*SetEventEv)(This,BOOL *bl0,BOOL *bl1,BYTE byEvent);
     Virtual void (*InitTCHN)(This,PVOID psTable);
     Virtual void (*PreProc)(This);
     Virtual void (*Processing)(This);
     Virtual void (*PostProc)(This);
	 Virtual BOOL (*EventHandler)(This,SMESSAGE *pMsg);
	 Virtual void (*SetInPinEvent)(This);
	 Virtual void (*SaveAlarmPin)(This);
	 Virtual void (*SendObsrveMsg)(This);
Public
     STIPARAM *pP;
	 WORD *m_pnIN;
	 WORD m_wOldIN;

	 BYTE m_byEvent;
	 BYTE m_byErEventCh;

     BOOL m_blTmSetState;
     BYTE m_bySetTimer;
	 BYTE m_byErEventHi;

	 BOOL m_blTmRemState;
     BYTE m_byRemTimer;
	 BYTE m_byErEventLo;

	 BOOL m_blChState;
     BYTE m_byChTimer;

	 BOOL m_blSHIL,m_blRHIL;
	 BOOL m_blSLOL,m_blRLOL;
	 DECLARE_IMPLEMENT_BASE(CTeleSensor)
}
DECLARE_DEFINITION(CTeleInd)
#endif
```

#### bnrtelesensor.h
```c
/********************************************************************
 * COPYRIGHT -- Kontora
 ********************************************************************
 * Program: bnrmain
 * File: bnraninput.h
 * Author: Abramenya
 * Created: January 19, 2009
 *******************************************************************/

#ifndef __TELESENSOR_H__
#define __TELESENSOR_H__
#include "typedefs.h"
#include "bnrdebug.h"
#include "bnrpob.h"
#include "bnrmessage.h"
#include "bnrcomputer.h"

Class CTeleSensor
{
	 void (*CCTeleSensor)(This);
	 void (*DCTeleSensor)(This);
Public
     void (*Init)(This,PVOID *psTable);
     void (*ObserveProc)(This);
	 //UINT (*GetW)(This,BYTE *pbyParam);
	 void (*CheckAlarm)(This);
	 BOOL (*SaveChange)(This,BYTE byEvent,WORD wValue,BOOL blAlarm);
	 BOOL (*SavePinState)(This,BYTE byEvent,WORD wValue);
	 void (*SendBroadcast)(This,SKPEVENT *pEV);
	 void (*SendSMessage)(This,BYTE byBox,BYTE byFor,BYTE byType);
	 void (*Switch)(This);
	 Virtual BOOL (*EventHandler)(This,SMESSAGE *pMsg);
     Virtual void (*InitTCHN)(This,PVOID psTable);
     Virtual void (*PreProc)(This);
     Virtual void (*Processing)(This);
	 Virtual void (*PostProc)(This);
	 Virtual void (*SaveAlarmPin)(This);
	 Virtual void (*SetInPinEvent)(This);
	 Virtual void (*SendObsrveMsg)(This);

Public
     STIPARAM *pP;
	 BOOL m_blSetAlarm;
     BYTE m_byID;
     BYTE m_byType;
	 BYTE m_byALC;
	 BYTE m_byOldEvent;
	 SHARDCOMPUTERTABLE *m_pPCT;
     CPin *m_pPN;
	 PVOID m_pvValue;
	 BOOL *m_pvAlValue;
     CComputer *m_pComputer;
	 DECLARE_IMPLEMENT
}
DECLARE_DEFINITION(CTeleSensor)
#endif
```

#### bnrtelesignal.h
```c
/********************************************************************
 * COPYRIGHT -- Kontora
 ********************************************************************
 * Program: bnrmain
 * File: bnraninput.h
 * Author: Abramenya
 * Created: January 19, 2009
 *******************************************************************/

#ifndef __TELESIGNAL_H__
#define __TELESIGNAL_H__
#include "typedefs.h"
#include "bnrtelesensor.h"
#include "bnrpin.h"
#define DEF_SET_PULSE 5
#define DEF_REM_PULSE 5
Class CTeleSignal
{
	 void (*CCTeleSignal)(This);
	 void (*DCTeleSignal)(This);
Public
     BYTE (*CheckTS)(This);
	 Virtual BOOL (*EventHandler)(This,SMESSAGE *pMsg);
	 Virtual void (*InitTCHN)(This,PVOID psTable);
     Virtual void (*PreProc)(This);
	 Virtual void (*Processing)(This);
     Virtual void (*PostProc)(This);
	 Virtual void (*SetInPinEvent)(This);
	 Virtual void (*SaveAlarmPin)(This);
	 Virtual void (*SendObsrveMsg)(This);
Public
     STSPARAM *pP;
	 BOOL *m_pbIN;
	 BOOL m_blFSignal;
     BOOL m_blTmSetState;
	 BOOL m_blTmRemState;
     BYTE m_bySetPulce;
	 BYTE m_byRemPulce;
	 DECLARE_IMPLEMENT_BASE(CTeleSensor)
}
DECLARE_DEFINITION(CTeleSignal)
#endif
```

#### multi.h
```c
/********************************************************************
 * COPYRIGHT -- Kontora
 ********************************************************************
 * Program: bnrmain
 * File: bnraninput.h
 * Author: Abramenya
 * Created: January 19, 2009
 *******************************************************************/

#ifndef __MULTI_H__
#define __MULTI_H__
#include "typedefs.h"
#include "single.h"
Class CMulti
{
	 void (*CCMulti)(This);
	 void (*DCMulti)(This);
Public
	 DECLARE_IMPLEMENT_BASE(CSingle)
}
DECLARE_DEFINITION(CMulti)
#endif
```

#### single.h
```c
/********************************************************************
 * COPYRIGHT -- Kontora
 ********************************************************************
 * Program: bnrmain
 * File: bnraninput.h
 * Author: Abramenya
 * Created: January 19, 2009
 *******************************************************************/

#ifndef __SINGLE_H__
#define __SINGLE_H__
#include "typedefs.h"
Class CSingle
{
	 void (*CCSingle)(This);
	 void (*DCSingle)(This);
Public
	 DECLARE_IMPLEMENT
}
DECLARE_DEFINITION(CSingle)
#endif
```

#### typedefs.h
```c
/********************************************************************
 * COPYRIGHT -- Kontora
 ********************************************************************
 * Program: bnrmain
 * File: typedefs.h
 * Author: Alex
 * Created: January 22, 2009
 *******************************************************************/
#ifndef __TYPED_H__
#define __TYPED_H__
#include "bnrconst.h"
#include "bnrdbout.h"
//Start Automat
enum _tagTIEvent
{
	EV_SET_HI=0,
	EV_REM_HI,
	EV_SET_LO,
	EV_REM_LO,
	EV_CHG_PR,
	EV_0T1_CH,
	EV_1T0_CH,
	EV_SAL_CH,
	EV_RAL_CH,
	EV_0T1_ST,
	EV_1T0_ST,
	EV_INI_CH,
	EV_ALP_CH,
	EV_ALS_CH,
	EV_CHK_CH,
};
enum _enTSParam
{
	EN_SET_PERIOD,
	EN_REM_PERIOD,
	EN_PIN_ALMODE,
};

enum _enCmdTypeParam
{
	CTR_TU,
	CTR_TR,
	CTR_OPEN,
	CTR_CLOSE,
	CTR_STOP,
};

#define S_BAD 0xFF
#define EXIT_D 0xFF
#define MSGIR_REQ              0x80
#define MC_UNKNOWN             0x7F
#define EV_UNKNOWN_REQ         (MC_UNKNOWN|MSGIR_REQ)
#define MAXNBVALUE             100
typedef unsigned char  TStateCode;
typedef unsigned char  TTask;
typedef unsigned char  TEvent;
typedef struct _tagTState
{
    TEvent m_vEvent;
    TTask* m_pvTask;
}TState;
typedef struct _tagTStateList
{
    TStateCode m_vStateCode;
    TState*    m_pvState;
}TStateList;
#define DECLARE_TASKCHAIN(Name) TTask          Name[]=
#define IMPORT_TASKCHAIN(Name)  extern TTask   Name[]
#define DECLARE_STATE(Name)     TState         Name[]=
#define IMPORT_STATE(Name)      extern TState  Name[]
#define DECLARE_STATELIST(Name) TStateList   Name[]=
#define IMPORT_STATELIST(Name)  extern TStateList  Name[]
//End Automat
#ifndef WIN32
 typedef UINT WORD;
 typedef UDINT DWORD;
 typedef UINT USHORT;
 typedef USINT BYTE;
 typedef void* PVOID;
 typedef BYTE* MESSAGE;
  typedef INT INT16;
#else
 #include <stdio.h>
 #include <stdlib.h>
#include <windows.h>
#include <malloc.h>
#include <string.h>
 #define MEM_alloc(X,Y) Y = malloc(X);
 #define MEM_free(X,Y)  free(Y);
 typedef unsigned char USINT;
 //typedef WORD UINT;
 typedef char SINT;
 typedef _int16 INT16;
 //typedef unsigned int WORD;

 typedef float REAL;
 typedef INT DINT;
 typedef unsigned long UDINT;
 typedef unsigned long DWORD;
 typedef unsigned char BYTE;
 typedef void* PVOID;
 typedef BYTE* MESSAGE;
 #define _GLOBAL
 #define _INIT
 #define _CYCLIC
 #define _EXIT
#endif
typedef BOOL (*PCLB)(PVOID,BYTE);
#define This PVOID pV
_GLOBAL void **pGlobalMemoryPointer;
_GLOBAL DWORD dwFL;
void CrateProcess(PVOID,SINT*,BYTE,BYTE);
#define FCREATE(X0,X1,X2,X3) CrateProcess(X0,X1,X2,X3);
void CrateTimer(PVOID);
void DeleteTimer(PVOID);
#define FCTIMER(X0) CrateTimer(X0);
#define FDTIMER(X0) DeleteTimer(X0);
void NEW(int nSize,void **pVoid);
void FREE(int nSize,void **pVoid);
#define New(X,Y) NEW(X,(void**)&Y)
#define Delete(X,Y) FREE(X,(void**)Y)
#define Public
#define Private
#define Protected
#define Virtual
#define Class typedef struct

#define DIP12_AVL(X) _GLOBAL BOOL  *blpValueDI##X##[DEV_MAX_DI_X20DM9371_PIN];
#define DIP2_AVL(X)  _GLOBAL UINT  *uipValueDI##X##[DEV_MAX_DI_X20DI2377_PIN];
#define DIP_AVL(X)   _GLOBAL BOOL  *blpValueDI##X##[DEV_MAX_DI_3DI477_PIN];
#define DOP_AVL(X)   _GLOBAL BOOL  *blpValueDO##X##[DEV_MAX_DO_3DO760_PIN];
#define DOP12_AVL(X) _GLOBAL BOOL  *blpValueDO##X##[DEV_MAX_DO_X20DM9322_PIN];
#define AIP4_AVL(X)  _GLOBAL UINT  *uipValueAI##X##[DEV_MAX_AI_X20AI4622_PIN];
#define AIP2_AVL(X)  _GLOBAL UINT  *uipValueAI##X##[DEV_MAX_AI_X20AI2622_PIN];
#define AIP_AVL(X)   _GLOBAL UINT  *uipValueAI##X##[DEV_MAX_AI_3AI375_PIN];
#define AOP_AVL(X)   _GLOBAL UINT  *uipValueAO##X##[DEV_MAX_AO_3AO775_PIN];
#define AOP4_AVL(X)  _GLOBAL UINT  *uipValueAO##X##[4];

#define DIP12_ALVL(X) _GLOBAL BOOL  *blpAlValueDI##X##[DEV_MAX_DI_X20DM9371_PIN];
#define DIP2_ALVL(X)  _GLOBAL BOOL  *blpAlValueDI##X##[DEV_MAX_DI_X20DI2377_PIN];
#define DOP12_ALVL(X) _GLOBAL BOOL  *blpAlValueDO##X##[DEV_MAX_DO_X20DM9322_PIN];
#define AIP4_ALVL(X)  _GLOBAL BOOL  *blpAlValueAI##X##[DEV_MAX_AI_X20AI4622_PIN];
#define AIP2_ALVL(X)  _GLOBAL BOOL  *blpAlValueAI##X##[DEV_MAX_AI_X20AI2622_PIN];
#define AOP4_ALVL(X)  _GLOBAL BOOL  *blpAlValueAO##X##[DEV_MAX_AO_X20AO4622_PIN];

#define DI_VL(X,Y)   _GLOBAL BOOL  blValueDI##X##_##Y##;
#define DIC_VL(X,Y)  _GLOBAL BOOL  uiValueDI##X##_##Y##;
#define DO_VL(X,Y)   _GLOBAL BOOL  blValueDO##X##_##Y##;
#define AI_VL(X,Y)   _GLOBAL INT16 uiValueAI##X##_##Y##;
#define AO_VL(X,Y)   _GLOBAL INT16 uiValueAO##X##_##Y##;

#define DI_ALVL(X,Y) _GLOBAL BOOL  blAlValueDI##X##_##Y##;
#define DO_ALVL(X,Y) _GLOBAL BOOL  blAlValueDO##X##_##Y##;
#define AI_ALVL(X,Y) _GLOBAL BOOL  blAlValueAI##X##_##Y##;
#define AO_ALVL(X,Y) _GLOBAL BOOL  blAlValueAO##X##_##Y##;

#define AI_ASVL(X)   _GLOBAL BOOL  blAsValueAI##X##;
#define AO_ASVL(X)   _GLOBAL BOOL  blAsValueAO##X##;
#define DI_ASVL(X)   _GLOBAL BOOL  blAsValueDI##X##;
#define DO_ASVL(X)   _GLOBAL BOOL  blAsValueDO##X##;

#define DI_SL(X) \
DI_VL(X,0)  DI_VL(X,1)  DI_VL(X,2)  DI_VL(X,3)  DI_VL(X,4)  DI_VL(X,5)  DI_VL(X,6)  DI_VL(X,7) \
DI_VL(X,8)  DI_VL(X,9)  DI_VL(X,10) DI_VL(X,11) DI_VL(X,12) DI_VL(X,13) DI_VL(X,14) DI_VL(X,15) \
DI_VL(X,16) DI_VL(X,17) DI_VL(X,18) DI_VL(X,19) DI_VL(X,20) DI_VL(X,21) DI_VL(X,22) DI_VL(X,23) \
DI_VL(X,24) DI_VL(X,25) DI_VL(X,26) DI_VL(X,27) DI_VL(X,28) DI_VL(X,29) DI_VL(X,30) DI_VL(X,31)
#define DI8_SL(X) DI_VL(X,0) DI_VL(X,1) DI_VL(X,2) DI_VL(X,3) DI_VL(X,4) DI_VL(X,5) DI_VL(X,6) DI_VL(X,7)
#define DO_SL(X)  DO_VL(X,0) DO_VL(X,1) DO_VL(X,2) DO_VL(X,3) DO_VL(X,4) DO_VL(X,5) DO_VL(X,6) DO_VL(X,7)

#define DI12_SL(X) DI_VL(X,0) DI_VL(X,1) DI_VL(X,2) DI_VL(X,3) DI_VL(X,4) DI_VL(X,5) DI_VL(X,6) DI_VL(X,7) DI_VL(X,8) DI_VL(X,9) DI_VL(X,10) DI_VL(X,11)
#define DIC2_SL(X) DIC_VL(X,0) DIC_VL(X,1)
#define DI12_ALSL(X) DI_ALVL(X,0) DI_ALVL(X,1) DI_ALVL(X,2) DI_ALVL(X,3) DI_ALVL(X,4) DI_ALVL(X,5) DI_ALVL(X,6) DI_ALVL(X,7) DI_ALVL(X,8) DI_ALVL(X,9) DI_ALVL(X,10) DI_ALVL(X,11)
#define DI2_ALSL(X) DI_ALVL(X,0) DI_ALVL(X,1)

#define DO12_SL(X)  DO_VL(X,0) DO_VL(X,1) DO_VL(X,2) DO_VL(X,3) DO_VL(X,4) DO_VL(X,5) DO_VL(X,6) DO_VL(X,7) DO_VL(X,8) DO_VL(X,9) DO_VL(X,10) DO_VL(X,11)
#define DO12_ALSL(X) DO_ALVL(X,0) DO_ALVL(X,1) DO_ALVL(X,2) DO_ALVL(X,3) DO_ALVL(X,4) DO_ALVL(X,5)  DO_ALVL(X,6) DO_ALVL(X,7) DO_ALVL(X,8) DO_ALVL(X,9) DO_ALVL(X,10) DO_ALVL(X,11)

#define AI_SL(X)  AI_VL(X,0) AI_VL(X,1) AI_VL(X,2) AI_VL(X,3) AI_VL(X,4) AI_VL(X,5) AI_VL(X,6) AI_VL(X,7)

#define AI2_SL(X) AI_VL(X,0) AI_VL(X,1)
#define AI4_SL(X) AI_VL(X,0) AI_VL(X,1) AI_VL(X,2) AI_VL(X,3)
#define AO4_SL(X) AO_VL(X,0) AO_VL(X,1) AO_VL(X,2) AO_VL(X,3)
#define AI4_ALSL(X) AI_ALVL(X,0) AI_ALVL(X,1) AI_ALVL(X,2) AI_ALVL(X,3)
#define AI2_ALSL(X) AI_ALVL(X,0) AI_ALVL(X,1)

#define AO4_ALSL(X) AO_ALVL(X,0) AO_ALVL(X,1) AO_ALVL(X,2) AO_ALVL(X,3)

#define AO_SL(X)  AO_VL(X,0) AO_VL(X,1) AO_VL(X,2) AO_VL(X,3) AO_VL(X,4) AO_VL(X,5) AO_VL(X,6) AO_VL(X,7)

//Connection
#define DI_CON(X,Y)  blpValueDI##X##[##Y##]   = &blValueDI##X##_##Y##;
#define DIC_CON(X,Y) uipValueDI##X##[##Y##]   = &uiValueDI##X##_##Y##;
#define DO_CON(X,Y)  blpValueDO##X##[##Y##]   = &blValueDO##X##_##Y##;
#define AI_CON(X,Y)  uipValueAI##X##[##Y##]   = &uiValueAI##X##_##Y##;
#define AO_CON(X,Y)  uipValueAO##X##[##Y##]   = &uiValueAO##X##_##Y##;

#define DI_ACN(X,Y)  blpAlValueDI##X##[##Y##] = &blAlValueDI##X##_##Y##;
#define DO_ACN(X,Y)  blpAlValueDO##X##[##Y##] = &blAlValueDO##X##_##Y##;
#define AI_ACN(X,Y)  blpAlValueAI##X##[##Y##] = &blAlValueAI##X##_##Y##;
#define AO_ACN(X,Y)  blpAlValueAO##X##[##Y##] = &blAlValueAO##X##_##Y##;

#define DI_CSL(X) \
DI_CON(X,0)  DI_CON(X,1)  DI_CON(X,2)  DI_CON(X,3)  DI_CON(X,4)  DI_CON(X,5)  DI_CON(X,6)  DI_CON(X,7) \
DI_CON(X,8)  DI_CON(X,9)  DI_CON(X,10) DI_CON(X,11) DI_CON(X,12) DI_CON(X,13) DI_CON(X,14) DI_CON(X,15) \
DI_CON(X,16) DI_CON(X,17) DI_CON(X,18) DI_CON(X,19) DI_CON(X,20) DI_CON(X,21) DI_CON(X,22) DI_CON(X,23) \
DI_CON(X,24) DI_CON(X,25) DI_CON(X,26) DI_CON(X,27) DI_CON(X,28) DI_CON(X,29) DI_CON(X,30) DI_CON(X,31)

#define DI12_CSL(X) DI_CON(X,0) DI_CON(X,1) DI_CON(X,2) DI_CON(X,3) DI_CON(X,4) DI_CON(X,5) DI_CON(X,6) DI_CON(X,7) DI_CON(X,8) DI_CON(X,9) DI_CON(X,10) DI_CON(X,11)
#define DIC2_CSL(X) DIC_CON(X,0) DIC_CON(X,1)
#define DO_CSL(X)   DO_CON(X,0) DO_CON(X,1) DO_CON(X,2) DO_CON(X,3) DO_CON(X,4) DO_CON(X,5) DO_CON(X,6) DO_CON(X,7)
#define DO12_CSL(X) DO_CON(X,0) DO_CON(X,1) DO_CON(X,2) DO_CON(X,3) DO_CON(X,4) DO_CON(X,5) DO_CON(X,6) DO_CON(X,7) DO_CON(X,8) DO_CON(X,9) DO_CON(X,10) DO_CON(X,11)
#define AI_CSL(X)   AI_CON(X,0) AI_CON(X,1) AI_CON(X,2) AI_CON(X,3) AI_CON(X,4) AI_CON(X,5) AI_CON(X,6) AI_CON(X,7)
#define AI4_CSL(X)  AI_CON(X,0) AI_CON(X,1) AI_CON(X,2) AI_CON(X,3)
#define AO4_CSL(X)  AO_CON(X,0) AO_CON(X,1) AO_CON(X,2) AO_CON(X,3)
#define AI2_CSL(X)  AI_CON(X,0) AI_CON(X,1)

#define DI12_ALCSL(X) DI_ACN(X,0) DI_ACN(X,1) DI_ACN(X,2) DI_ACN(X,3) DI_ACN(X,4) DI_ACN(X,5) DI_ACN(X,6) DI_ACN(X,7) DI_ACN(X,8) DI_ACN(X,9) DI_ACN(X,10) DI_ACN(X,11)
#define DI2_ALCSL(X)  DI_ACN(X,0) DI_ACN(X,1)

#define DO12_ALCSL(X) DO_ACN(X,0) DO_ACN(X,1) DO_ACN(X,2) DO_ACN(X,3) DO_ACN(X,4) DO_ACN(X,5) DO_ACN(X,6) DO_ACN(X,7) DO_ACN(X,8) DO_ACN(X,9) DO_ACN(X,10) DO_ACN(X,11)
#define AI4_ALCSL(X ) AI_ACN(X,0) AI_ACN(X,1) AI_ACN(X,2) AI_ACN(X,3)
#define AI2_ALCSL(X ) AI_ACN(X,0) AI_ACN(X,1)
#define AO4_ALCSL(X ) AO_ACN(X,0) AO_ACN(X,1) AO_ACN(X,2) AO_ACN(X,3)

#define AO_CSL(X)  AO_CON(X,0) AO_CON(X,1) AO_CON(X,2) AO_CON(X,3) AO_CON(X,4) AO_CON(X,5) AO_CON(X,6) AO_CON(X,7)
#define DI_INI12(X,Y) for(i=0;i<11;i++) *blpValueDI##X##[i] = Y;
#define DIC_INI2(X,Y) for(i=0;i<2;i++) *uipValueDI##X##[i] = Y;

#define AI_ALIN4(X,Y)  for(i=0;i<4;i++)  *blpAlValueAI##X##[i] = Y;
#define AO_ALOT4(X,Y)  for(i=0;i<4;i++)  *blpAlValueAO##X##[i] = Y;
#define AI_ALIN2(X,Y)  for(i=0;i<2;i++)  *blpAlValueAI##X##[i] = Y;
#define DI_ALIN12(X,Y) for(i=0;i<11;i++) *blpAlValueDI##X##[i] = Y;
#define DI_ALIN2(X,Y) for(i=0;i<2;i++) *blpAlValueDI##X##[i] = Y;
#define DO_ALIN12(X,Y) for(i=0;i<11;i++) *blpAlValueDO##X##[i] = Y;

#define DI_INI(X,Y) for(i=0;i<20;i++) *blpValueDI##X##[i] = Y;
#define DI8_INI(X,Y)for(i=0;i<7;i++) *blpValueDI##X##[i] = Y;
#define DECLARE_DEFINITION(X)X; void X##_CreateClass(##X *pM);void X##_DestroyClass(##X *pM);
#define DECLARE_IMPLEMENT_BASE(X)  \
	X m_n##X; \
	X *pBase; \
	PVOID pThis; \
	PVOID pChld;
#define DECLARE_IMPLEMENT  \
	PVOID pBase; \
	PVOID pThis; \
	PVOID pChld;
#define DECLARE_SINGLE_CREATE(X) \
	void X##_CreateClass(##X *pM)\
	{ \
    pM->pBase = NULL; \
	pM->pThis = pM; \
	pM->pChld = pM; \
	pM->C##X = X##_##X; \
    pM->D##X = X##_D##X; \
	pM->C##X(pM); \
	}; \
	void X##_DestroyClass(##X *pM) \
	{	\
     X##_D##X##(pM); \
	};
#define DECLARE_MULTI_CREATE(X,Y) \
	void X##_CreateClass(##X *pM)\
	{ \
	pM->pBase = &pM->m_n##Y; \
	pM->pThis = pM; \
	pM->pChld = NULL; \
	InitObject(Y,&pM->m_n##Y) \
	pM->m_n##Y##.pChld = pM; \
	pM->C##X = X##_##X; \
	pM->D##X = X##_D##X; \
	pM->C##X(pM); \
	}; \
	void X##_DestroyClass(##X *pM) \
	{ \
	 X##_D##X##(pM); \
	};
#define DECLARE_SINGLE_OPEN(X) \
	X *pT = pV; \
	X *pC = pT->pChld;
#define DECLARE_MULTI_OPEN(X,Y) \
	X *pT = pV; \
	Y *pB = pT->pBase; \
    PVOID *pC = pT->pChld;
#define DECLARE_REGISTRATION(X,Y) pT->Y = X##_##Y;
#define DECLARE_VIRTUAL_FUNC(X,Y) pT->Y = X##_##Y; pB->Y = pT->Y;
#define DECLARE_VIRTUAL1_FUNC(X,Y) pT->Y = X##_##Y; pB->pBase->Y = pT->Y;
#define InitObject(X,Y) X##_CreateClass(Y);
#define DeleteObject(X) if(X!=0)Delete(sizeof(*X),X);X=0;
#define DestroyObject(X,Y) if(Y!=NULL){X##_DestroyClass(Y);Delete(sizeof(*((X*)Y)),Y);}
#define DestroyObjectB(X,Y) if(Y!=NULL){X##_DestroyClass(Y);}
#define DESTROY Delete(sizeof(*pT),pT);
#endif
```

#### bnrcomvs1.h
```c
/********************************************************************
 * COPYRIGHT -- Kontora
 ********************************************************************
 * Program: bnrmain
 * File: bnraninput.h
 * Author: Abramenya
 * Created: January 19, 2009
 *******************************************************************/

#ifndef __COMVS1_H__
#define __COMVS1_H__
#include "typedefs.h"
#include "bnrmessage.h"
#include "bnrdebug.h"
#include "bnrcyclicsystem.h"

#ifndef WIN32
//#include <DVFrame.h>
#endif
#define BUFF_SZ_VS1 0x3ff
Class CComVS1
{
	 void (*CCComVS1)(This);
	 void (*DCComVS1)(This);
Public
     //Connection Disconnection Procedure
     void (*Init)(This,SARMINTERFACE *pArm);
Private
	 void (*Close)(This);
     void (*InitSRV)(This);
	 void (*Enable)(This);
	 void (*Disable)(This);
	 BOOL (*Open)(This);
     BOOL (*SendMessage)(This,SMESSAGE *pMsg);
	 BOOL (*GetMessage)(This,SMESSAGE *pMsg);
	 void (*ReceiveThread)(This);
	 void (*SendThread)(This);
	 void (*SynBuff)(This);
	 BOOL (*MakeMsgData)(This,SMESSAGE *pMsg);
	 BOOL (*CopyMessage)(This,WORD wLen,SMESSAGE *pMsg);
	 BYTE (*CreateCRC)(This,BYTE *pMsg,BYTE byLen);
	 void (*SendSMessage)(This,BYTE byBox,BYTE byFor,BYTE byType);
	 BOOL (*Connect)(This);
	 BOOL (*Disconnect)(This);
	 void (*SetPortSett)(This);
     Virtual BOOL (*EventHandler)(This,SMESSAGE *pMsg);
     Virtual void (*CyclicProc)(This);
Private
	 SINT m_chStringDevice[50];
     SINT m_chStringMode[50];
	 SINT m_chStringNewMode[50];
     UINT m_StatusOpen;
	 UINT m_StatusClose;
	 UINT m_StatusWrite;
	 UINT m_StatusRead;
	 UINT m_StatusGetBuffer;
	 UINT m_StatusReleaseBuffer;
	 UINT m_StatusReleaseOutputBuffer;
	 UINT m_SendBufferLength;
	 UINT m_ReadBufferLength;
	 UINT m_Error;
	 UINT w_lMsgLen;

	 USINT m_SendBuffer[300];
	 USINT m_ReadBuffer[300];
	 USINT pb_mBoxDoTextRead[120];
	 BYTE pb_mBoxCont[BUFF_SZ_VS1];
	 WORD w_mBoxSize;
	 WORD w_mBoxCSize;
	 WORD w_mBoxWrite;
	 WORD w_mBoxRead;
	 WORD m_sSize;
     WORD w_lLength;
	 WORD InByteCount_DATA;

	 BYTE m_byType;
	 BYTE m_byRate;
	 BOOL m_blMsgFind;
     STCPADDR m_stTcpAddr;
	 BYTE m_bSrvState;
	 BYTE m_bCliState;
	 SMESSAGE m_sMsg;
	 CMTimer m_nConnTMR;
	 SARMINTERFACE *m_pArm;
	 DECLARE_IMPLEMENT_BASE(CCyclicSystem)
}
DECLARE_DEFINITION(CComVS1)
#endif
```

#### bnrcomvs0.c
```c
/********************************************************************
 * COPYRIGHT -- Kontora
 ********************************************************************
 * Program: bnrmain
 * File: bnrlsens.c
 * Author: Abramenya
 * Created: January 19, 2009
 *******************************************************************/

#include "bnrcomvs0.h"
#ifdef _DEFAULT_INCLUDES
 #include <AsDefault.h>
#endif
extern SINT *chPortType[];
extern SINT *chPortRate[];
extern SINT *chPortParity[];
extern SINT *chPortData[];
extern SINT *chPortStop[];
_GLOBAL FRM_xopen_typ m_sXOpenVS0;
_GLOBAL XOPENCONFIG   m_sConfigVS0;
_GLOBAL FRM_gbuf_typ  m_sFrameBuffVS0;
_GLOBAL FRM_rbuf_typ  m_sRBuffVS0;
_GLOBAL FRM_write_typ m_sSendVS0;
_GLOBAL FRM_read_typ  m_sReccVS0;
_GLOBAL FRM_close_typ m_sCloseVS0;
_GLOBAL FRM_robuf_typ m_sRobuffVS0;
#ifndef WIN32
_GLOBAL FRM_mode_typ FrameModeStructVS0;
#endif

void CComVS0_Init(This,SARMINTERFACE *pArm)
{
    DECLARE_MULTI_OPEN(CComVS0,CCyclicSystem)
    //#ifdef WIN32
	//m_nCommServer = pT;
    //#endif
	pT->m_pArm = pArm;
	FDEFINE(DEV_RSVS0MMD_BOX_ID,1024);
	FDEFINE(DEV_RSVBS0_BOX_ID,1024);
	pB->SetBoxID(pB,DEV_RSVS0MMD_BOX_ID);

	InitObject(CMTimer,&pT->m_nConnTMR);
	pT->m_nConnTMR.SetTimer(&pT->m_nConnTMR,DIR_PHTOPH,DIR_PHTOPH,EV_TMR_SRR_REQ,0,0,DEV_RSVS0MMD_BOX_ID);

	pT->m_blMsgFind = FALSE;
	pT->m_byType = pArm->byType;
	pT->m_byRate = pArm->byPortRate;
	pT->InByteCount_DATA = 0;

	strcpy(pT->m_chStringMode, chPortType[pT->m_pArm->byType]);
	strcat(pT->m_chStringMode,", ");
	strcat(pT->m_chStringMode, chPortRate[pT->m_pArm->byPortRate]);
	strcat(pT->m_chStringMode,", ");
	strcat(pT->m_chStringMode, chPortParity[pT->m_pArm->stTcpAddr.byAddr0]);
	strcat(pT->m_chStringMode,", ");
	strcat(pT->m_chStringMode, chPortData[pT->m_pArm->stTcpAddr.byAddr1]);
	strcat(pT->m_chStringMode,", ");
	strcat(pT->m_chStringMode, chPortStop[pT->m_pArm->stTcpAddr.byAddr2]);

	strcpy(pT->m_chStringDevice, "IF4.ST1");
	#ifdef DEB_CComVS0
	Info("\n(__)CTCPS::>Create %s.Device: %s Mode: %s",
	chPortType[pT->m_byType],pT->m_chStringDevice,pT->m_chStringMode);
	#endif
	pT->SynBuff(pT);
    pT->InitSRV(pT);
	//pT->m_nConnTMR.OnTimer(&pT->m_nConnTMR,200);
	pT->m_StatusWrite = 0;
	pT->m_bSrvState = DRV_ST_CONN;
	pT->m_bCliState = DRV_ST_CONN;
}
void CComVS0_SetPortSett(This)
{
    DECLARE_MULTI_OPEN(CComVS0,CCyclicSystem)
    strcpy(pT->m_chStringDevice, "IF4.ST1");
	memset(pT->m_chStringNewMode,0,sizeof(pT->m_chStringNewMode));

	strcpy(pT->m_chStringNewMode, chPortType[pT->m_pArm->byType]);
	strcat(pT->m_chStringNewMode,", ");
	strcat(pT->m_chStringNewMode, chPortRate[pT->m_pArm->byPortRate]);
	strcat(pT->m_chStringNewMode,", ");
	strcat(pT->m_chStringNewMode, chPortParity[pT->m_pArm->stTcpAddr.byAddr0]);
	strcat(pT->m_chStringNewMode,", ");
	strcat(pT->m_chStringNewMode, chPortData[pT->m_pArm->stTcpAddr.byAddr1]);
	strcat(pT->m_chStringNewMode,", ");
	strcat(pT->m_chStringNewMode, chPortStop[pT->m_pArm->stTcpAddr.byAddr2]);
    #ifndef WIN32
    FrameModeStructVS0.ident  = m_sXOpenVS0.ident;
    FrameModeStructVS0.mode   = (UDINT)pT->m_chStringNewMode;
    FrameModeStructVS0.enable = 1;
    FRM_mode(&FrameModeStructVS0);
    #endif
}
void CComVS0_SynBuff(This)//CANOpen
{
    DECLARE_MULTI_OPEN(CComVS0,CCyclicSystem)
	pT->w_mBoxSize  = BUFF_SZ_VS0;
    pT->w_mBoxCSize = BUFF_SZ_VS0;
	pT->w_mBoxWrite = 0;
	pT->w_mBoxRead  = 0;
	pT->m_sSize     = 0;
	pT->w_lLength   = 0;
	pT->w_lMsgLen   = 0;
	memset(&pT->pb_mBoxCont[0],0,10);
	#ifdef DEB_CComVS0
	Info("\n(__)CTCPS::>Synchro.");
    #endif
}
//_GLOBAL FRM_xopen_typ FrameXOpenStruct;
//_GLOBAL XOPENCONFIG XOpenConfigStruct;
void CComVS0_InitSRV(This)
{
    DECLARE_MULTI_OPEN(CComVS0,CCyclicSystem)
	//Server Init
    m_sConfigVS0.idle     = 10;
    m_sConfigVS0.delimc   = 0;
    m_sConfigVS0.delim[0] = 0;
	m_sConfigVS0.delim[1] = 0;
	m_sConfigVS0.tx_cnt   = 2;
	m_sConfigVS0.rx_cnt   = 2;
	m_sConfigVS0.tx_len   = 256;
	m_sConfigVS0.rx_len   = 256;
	m_sConfigVS0.argc     = 0;
	m_sConfigVS0.argv     = 0;

	strcpy(pT->m_chStringMode, "RS232, 1200, N, 8, 1");
	m_sXOpenVS0.device    = (UDINT) pT->m_chStringDevice;
	m_sXOpenVS0.mode      = (UDINT) pT->m_chStringMode;
    m_sXOpenVS0.config    = (UDINT)&m_sConfigVS0;
	m_sXOpenVS0.enable    = 1;
	pT->m_StatusOpen   = 0;
    #ifndef WIN32
	pT->m_nConnTMR.OnTimer(&pT->m_nConnTMR,30);
    #else
	pT->m_nConnTMR.OnTimer(&pT->m_nConnTMR,30);
	//pT->Open(pT);
    #endif
}
_GLOBAL INT nOPEN,nCLOSE;

BOOL CComVS0_Open(This)
{
    DECLARE_MULTI_OPEN(CComVS0,CCyclicSystem)
	SHORTMESSAGE m_sMsg;
    if(pT->m_StatusOpen==0)
	{
	#ifndef WIN32
	FRM_xopen(&m_sXOpenVS0);
    #endif
	if(m_sXOpenVS0.status==0)
	{
	 nOPEN++;
	 m_sReccVS0.ident      = m_sXOpenVS0.ident;
	 m_sSendVS0.ident      = m_sXOpenVS0.ident;
	 m_sCloseVS0.ident     = m_sXOpenVS0.ident;
	 m_sFrameBuffVS0.ident = m_sXOpenVS0.ident;
	 m_sRBuffVS0.ident     = m_sXOpenVS0.ident;
	 m_sReccVS0.buffer	    = (UDINT)&pT->m_ReadBuffer[0];
	 m_sSendVS0.buffer     = (UDINT)&pT->m_SendBuffer[0];
	 m_sFrameBuffVS0.buffer= m_sSendVS0.buffer;
	 m_sRBuffVS0.buffer    = m_sReccVS0.buffer;
	 m_sReccVS0.enable     = 1;
	 m_sSendVS0.enable     = 1;
	 m_sCloseVS0.enable    = 1;
	 m_sFrameBuffVS0.enable= 1;
	 m_sRBuffVS0.enable    = 1;
	 pT->m_StatusOpen   = 1;
	 pT->m_StatusWrite  = 0;
	 //pT->SendSMessage(pT,DEV_KPMDL_BOX_ID,DIR_PHTOKP,PH_CALL_REQ);
	 return TRUE;
	}
 	}
	return FALSE;
}
void CComVS0_Enable(This)
{
	DECLARE_MULTI_OPEN(CComVS0,CCyclicSystem)
	m_sXOpenVS0.enable = 1;
}
void CComVS0_Disable(This)
{
	DECLARE_MULTI_OPEN(CComVS0,CCyclicSystem)
	m_sXOpenVS0.enable = 0;
}
void CComVS0_Close(This)
{
    DECLARE_MULTI_OPEN(CComVS0,CCyclicSystem)
	m_sCloseVS0.enable = 1;
	FRM_close(&m_sCloseVS0);
}
BOOL CComVS0_SendMessage(This,SMESSAGE *pMsg)
{
	DECLARE_MULTI_OPEN(CComVS0,CCyclicSystem)
	BOOL res = TRUE;
	if(pT->m_StatusOpen==1)
	{
	 FRM_gbuf(&m_sFrameBuffVS0);
     m_sSendVS0.buflng = pMsg->m_swLen-9;
	 memcpy(m_sSendVS0.buffer, &pMsg->m_sbyInfo[0],m_sSendVS0.buflng);
	 FRM_write(&m_sSendVS0);
	 pT->m_StatusWrite  = m_sSendVS0.status;
	 if(pT->m_StatusWrite==0) res = TRUE;else res = FALSE;
	}
	return res;
}
_GLOBAL INT nSNDVS0;
_GLOBAL INT nSendThreadVS0;
void CComVS0_SendThread(This)
{
    DECLARE_MULTI_OPEN(CComVS0,CCyclicSystem)
	nSendThreadVS0++;
    //if(pT->m_StatusWrite==0)
	if(pT->m_StatusOpen==1)
    {
	 if(FGET(DEV_RSBUF_BOX_ID,&pT->m_sMsg))
	 {
	  //Info("\n(__)CRSVO::>TX:%M",&pT->m_sMsg);
	  if(pT->m_sMsg.m_swLen<=256)
	  {
	   nSNDVS0++;
       pT->SendMessage(pT,&pT->m_sMsg);
	  }//else
	    //Info("\n(__)CRSVO::>Wery Long Message!");
	 }
	}
 	 //else
 	 //{
 	 // #ifdef DEB_CComVS0
 	 // ///Info("\n(__)Wait.");
 	 // #endif
 	 //}
}
_GLOBAL INT nGETL1VS0;
BOOL CComVS0_GetMessage(This,SMESSAGE *pMsg)
{
    DECLARE_MULTI_OPEN(CComVS0,CCyclicSystem)
	BYTE i,*pBuff;
	BOOL res=FALSE;
	SMESSAGE csM;
	if(pT->m_StatusOpen==1)
	{
	FRM_read(&m_sReccVS0);
	pT->m_StatusRead       = m_sReccVS0.status;
	if(pT->m_StatusRead==0)
	{
	 pT->m_ReadBufferLength = m_sReccVS0.buflng;
	 pBuff                  = m_sReccVS0.buffer;
	 /*
	 csM.m_sbyInfo[0] = 0x7e;
	 csM.m_sbyInfo[1] = 'A';
	 csM.m_sbyInfo[2] = 'l';
	 csM.m_sbyInfo[3] = 'e';
	 csM.m_sbyInfo[4] = 'x';
	 csM.m_sbyInfo[5] = 'a';
	 csM.m_sbyInfo[6] = 'n';
	 csM.m_sbyInfo[7] = 'd';
	 csM.m_sbyInfo[8] = 'e';
	 csM.m_sbyInfo[9] = 'r';
	 csM.m_sbyInfo[10] = 0xe7;
	 */

	 //memcpy(&csM.m_sbyInfo[0],m_sReccVS0.buffer,pT->m_ReadBufferLength);
	 //csM.m_swLen = 9 + pT->m_ReadBufferLength;
	 //Info("\n(__)CRSVO::>MSG:%M",&csM);

	 //m_sRBuffVS0.buffer = m_sReccVS0.buffer;
	 //m_sRBuffVS0.buflng = pT->m_ReadBufferLength;
	 //FRM_rbuf(&m_sRBuffVS0);
	 //res = TRUE;
	 //nGETL1++;
	 //Info("\nMSG::>");
	 //csM.m_swLen = pT->m_ReadBufferLength+9;
	 for( i=0;i<pT->m_ReadBufferLength;i++)
	 {
	  pT->pb_mBoxCont[pT->w_mBoxWrite] = pBuff[i];
      //Info(" %b",&pT->pb_mBoxCont[pT->w_mBoxWrite]);
	  //printf(" %c",pT->pb_mBoxCont[pT->w_mBoxWrite]);
      pT->w_mBoxWrite = (pT->w_mBoxWrite + 1) & BUFF_SZ_VS0;
	 }
	 //FPUT(DEV_RSBUF_BOX_ID,(BYTE*)&csM);
	 pT->w_mBoxSize -= pT->m_ReadBufferLength;
	 pT->m_sSize     = pT->w_mBoxCSize-pT->w_mBoxSize;
	 //Info("\nRD::>%b PRD::>%w PWD::>%w FND::>%b",&pT->pb_mBoxCont[pT->w_mBoxRead],&pT->w_mBoxRead,&pT->w_mBoxWrite,&pT->m_blMsgFind);
	 if ((pT->pb_mBoxCont[pT->w_mBoxRead]==0x3d))
	 {
		 pT->m_blMsgFind = TRUE;
		 if(res = pT->MakeMsgData(pT,pMsg))
		 {
			 pT->m_blMsgFind = FALSE;
			 res = TRUE;
		 }
	 }else
		 pT->SynBuff(pT);
	 m_sRBuffVS0.buffer = m_sReccVS0.buffer;
	 m_sRBuffVS0.buflng = pT->m_ReadBufferLength;
	 FRM_rbuf(&m_sRBuffVS0);
     }
	}
	return res;
}
BOOL CComVS0_MakeMsgData(This,SMESSAGE *pMsg)
{
    DECLARE_MULTI_OPEN(CComVS0,CCyclicSystem)
	WORD lLen,i,nCM=0;
	BOOL res = FALSE;
	lLen = 1;
	pT->w_lMsgLen = pT->w_lMsgLen + pT->m_ReadBufferLength;
	if (pT->w_lMsgLen>BUFF_SZ_VS0) {pT->SynBuff(pT);return res;}
    for (i=1;i<pT->w_lMsgLen-1;i++)
	{
	 lLen++;
	 if (pT->pb_mBoxCont[(pT->w_mBoxRead+i)& BUFF_SZ_VS0]==0x2e) nCM++;
	 if (nCM>1){pT->SynBuff(pT);return res;}
	 if (lLen>300) {pT->SynBuff(pT);return res;}
     if (pT->pb_mBoxCont[(pT->w_mBoxRead+i)& BUFF_SZ_VS0]==0x3d)
     {
	  pT->CopyMessage(pT,lLen,pMsg);
	  //pT->SynBuff(pT);
	  pT->w_lMsgLen = 0;
	  return TRUE;
	 }
	}
	return res;
}
BOOL CComVS0_CopyMessage(This,WORD wLen,SMESSAGE *pMsg)
{
    DECLARE_MULTI_OPEN(CComVS0,CCyclicSystem)
	INT i,j=0;BYTE byCRC;
	BOOL blCRC;
	for(i=0;i<wLen;i++)
	{
 	 if ((i!=0)&&(i!=wLen-1)){pMsg->m_sbyInfo[j]=pT->pb_mBoxCont[pT->w_mBoxRead];j++;}
	 pT->w_mBoxSize =(pT->w_mBoxSize+1)& BUFF_SZ_VS0;
	 pT->w_mBoxRead=(pT->w_mBoxRead+1)& BUFF_SZ_VS0;
	 //Info(" %b",&pMsg->m_sbyInfo[i]);
	 //printf(" %x",pMsg->m_sbyInfo[i]);
	}
	pMsg->m_sbyInfo[j++] = 0x00;
	pT->w_mBoxRead=(pT->w_mBoxRead-1)& BUFF_SZ_VS0;
	pT->m_sSize = (pT->w_mBoxCSize-pT->w_mBoxSize) & BUFF_SZ_VS0;
	pMsg->m_swLen         = j+9;
	pMsg->m_sbyFrom       = DIR_PHMDL;
	pMsg->m_sbyFor        = DIR_PHTOMS;
	pMsg->m_sbyIntType    = 0;
	pMsg->m_sbyServerID   = 0;
	pMsg->m_sbyType       = PH_VS0_REQ;
	pMsg->m_sbyDirection  = 0;
	pMsg->m_sbySensor     = 0;
	return TRUE;
}
BYTE CComVS0_CreateCRC(This,BYTE *pMsg,BYTE byLen)
{
	DECLARE_MULTI_OPEN(CComVS0,CCyclicSystem)
	BYTE i,sum = 0;
	for(i=0;i<=byLen-1;i++)sum += pMsg[i];
	return sum;
}
_GLOBAL INT nReceiveThreadVS0;
void CComVS0_ReceiveThread(This)
{
    DECLARE_MULTI_OPEN(CComVS0,CCyclicSystem)
	nReceiveThreadVS0++;
	#ifndef WIN32
	if(pT->GetMessage(pT,&pT->m_sMsg)==TRUE)
	{
	 //Info("\n(__)CRSVO::>RX:%M",&pT->m_sMsg);
	 FPUT(DEV_MSMDL_BOX_ID,(BYTE*)&pT->m_sMsg);
		//FPUT(DEV_RSBUF_BOX_ID,(BYTE*)&pT->m_sMsg);
	}
    #endif
}
_GLOBAL INT nRSEventHandlerVS0,nCheckOpenVS0,nWatchOpenVS0;
BOOL CComVS0_EventHandler(This,SMESSAGE *pMsg)
{
    DECLARE_MULTI_OPEN(CComVS0,CCyclicSystem)
	switch(pMsg->m_sbyFor)
	{
	  case DIR_101TOPH:
	       #ifdef DEB_CComVS0
		   Info("\n(__)CRSVO::>OUTP::%M",pMsg);
		   #endif
		   FPUT(DEV_RSBUF_BOX_ID,pMsg);
	  break;
	  case DIR_PHTOPH:
	       if (pMsg->m_sbyType==EV_TMR_SRR_REQ)
		   {
		   	//if(pT->m_StatusOpen==0)
			{
			 nCheckOpenVS0++;
 		     pT->Open(pT);
			}
			pT->m_nConnTMR.OnTimer(&pT->m_nConnTMR,30);
		   }
	  break;
      case DIR_KPTOPH:
	       if (pMsg->m_sbyType==PH_CLOSE_PORT_REQ)
		   {
            //pT->Close(pT);
		   }
		   if(pMsg->m_sbyType==PH_INIT_PORT_REQ)
		   {
             pT->SetPortSett(pT);
		   }
	  break;
	  default:
	  break;
	}
	return TRUE;
}
void CComVS0_Connect(This)
{
    DECLARE_MULTI_OPEN(CComVS0,CCyclicSystem)
    SHORTMESSAGE m_sMsg;
	m_sMsg.m_swLen        = 9;
	m_sMsg.m_sbyFrom      = DIR_PHMDL;
	m_sMsg.m_sbyFor       = DIR_PHTO101P;
	m_sMsg.m_sbyIntType   = 0;
	m_sMsg.m_sbyServerID  = 0;
	m_sMsg.m_sbyType      = PH_CONN_IND;
	m_sMsg.m_sbyDirection = 0;
	m_sMsg.m_sbySensor    = 0;
	FPUT(DEV_101MD_BOX_ID,(BYTE*)&m_sMsg);
    #ifdef DEB_CComVS0
	Info("\n(__)CRSVO::>OUTT::%M",&m_sMsg);
    #endif
}
void CComVS0_SendSMessage(This,BYTE byBox,BYTE byFor,BYTE byType)
{
    DECLARE_MULTI_OPEN(CComVS0,CCyclicSystem)
    SHORTMESSAGE m_sMsg;
	m_sMsg.m_swLen        = 9;
	m_sMsg.m_sbyFrom      = DIR_PHMDL;
	m_sMsg.m_sbyFor       = byFor;
	m_sMsg.m_sbyIntType   = 0;
	m_sMsg.m_sbyServerID  = 0;
	m_sMsg.m_sbyType      = byType;
	m_sMsg.m_sbyDirection = 0;
	m_sMsg.m_sbySensor    = 0;
	FPUT(byBox,(BYTE*)&m_sMsg);
    #ifdef DEB_CComVS0
	Info("\n(__)CRSVO::>OUTT::%M",&m_sMsg);
    #endif
}
void CComVS0_Disconnect(This)
{
    DECLARE_MULTI_OPEN(CComVS0,CCyclicSystem)
    SHORTMESSAGE m_sMsg;
	m_sMsg.m_swLen        = 9;
	m_sMsg.m_sbyFrom      = DIR_PHMDL;
	m_sMsg.m_sbyFor       = DIR_PHTO101P;
	m_sMsg.m_sbyIntType   = 0;
	m_sMsg.m_sbyServerID  = 0;
	m_sMsg.m_sbyType      = PH_DISC_IND;
	m_sMsg.m_sbyDirection = 0;
	m_sMsg.m_sbySensor    = 0;
	FPUT(DEV_101MD_BOX_ID,(BYTE*)&m_sMsg);
    #ifdef DEB_CComVS0
	Info("\n(__)CRSVO::>OUTT::%M",&m_sMsg);
    #endif
}
void CComVS0_CyclicProc(This)
{
    DECLARE_MULTI_OPEN(CComVS0,CCyclicSystem)
	pT->ReceiveThread(pT);
}
void CComVS0_CComVS0(This)
{
    DECLARE_MULTI_OPEN(CComVS0,CCyclicSystem)
	DECLARE_REGISTRATION(CComVS0,Init)
	DECLARE_REGISTRATION(CComVS0,InitSRV)
	DECLARE_REGISTRATION(CComVS0,SendMessage)
	DECLARE_REGISTRATION(CComVS0,GetMessage)
    DECLARE_REGISTRATION(CComVS0,Close)
	DECLARE_REGISTRATION(CComVS0,Disable)
	DECLARE_REGISTRATION(CComVS0,Enable)
	DECLARE_REGISTRATION(CComVS0,Open)
	DECLARE_REGISTRATION(CComVS0,ReceiveThread)
	DECLARE_REGISTRATION(CComVS0,SendThread)
	DECLARE_REGISTRATION(CComVS0,SynBuff)
	DECLARE_REGISTRATION(CComVS0,MakeMsgData)
	DECLARE_REGISTRATION(CComVS0,CopyMessage)
	DECLARE_REGISTRATION(CComVS0,CreateCRC)
	DECLARE_REGISTRATION(CComVS0,Connect)
	DECLARE_REGISTRATION(CComVS0,Disconnect)
	DECLARE_REGISTRATION(CComVS0,SendSMessage)
	DECLARE_REGISTRATION(CComVS0,SetPortSett)
	DECLARE_VIRTUAL_FUNC(CComVS0,EventHandler)
	DECLARE_VIRTUAL_FUNC(CComVS0,CyclicProc)
}

void CComVS0_DCComVS0(This)
{
	DECLARE_MULTI_OPEN(CComVS0,CCyclicSystem)
	//DESTROY
}

DECLARE_MULTI_CREATE(CComVS0,CCyclicSystem)
```

#### bnrcomvs0.h
```c
/********************************************************************
 * COPYRIGHT -- Kontora
 ********************************************************************
 * Program: bnrmain
 * File: bnraninput.h
 * Author: Abramenya
 * Created: January 19, 2009
 *******************************************************************/

#ifndef __COMVS0_H__
#define __COMVS0_H__
#include "typedefs.h"
#include "bnrmessage.h"
#include "bnrdebug.h"
#include "bnrcyclicsystem.h"

#ifndef WIN32
//#include <DVFrame.h>
#endif
#define BUFF_SZ_VS0 0x3ff
Class CComVS0
{
	 void (*CCComVS0)(This);
	 void (*DCComVS0)(This);
Public
     //Connection Disconnection Procedure
     void (*Init)(This,SARMINTERFACE *pArm);
Private
	 void (*Close)(This);
     void (*InitSRV)(This);
	 void (*Enable)(This);
	 void (*Disable)(This);
	 BOOL (*Open)(This);
     BOOL (*SendMessage)(This,SMESSAGE *pMsg);
	 BOOL (*GetMessage)(This,SMESSAGE *pMsg);
	 void (*ReceiveThread)(This);
	 void (*SendThread)(This);
	 void (*SynBuff)(This);
	 BOOL (*MakeMsgData)(This,SMESSAGE *pMsg);
	 BOOL (*CopyMessage)(This,WORD wLen,SMESSAGE *pMsg);
	 BYTE (*CreateCRC)(This,BYTE *pMsg,BYTE byLen);
	 void (*SendSMessage)(This,BYTE byBox,BYTE byFor,BYTE byType);
	 BOOL (*Connect)(This);
	 BOOL (*Disconnect)(This);
	 void (*SetPortSett)(This);
     Virtual BOOL (*EventHandler)(This,SMESSAGE *pMsg);
     Virtual void (*CyclicProc)(This);
Private
	 SINT m_chStringDevice[50];
     SINT m_chStringMode[50];
	 SINT m_chStringNewMode[50];
     UINT m_StatusOpen;
	 UINT m_StatusClose;
	 UINT m_StatusWrite;
	 UINT m_StatusRead;
	 UINT m_StatusGetBuffer;
	 UINT m_StatusReleaseBuffer;
	 UINT m_StatusReleaseOutputBuffer;
	 UINT m_SendBufferLength;
	 UINT m_ReadBufferLength;
	 UINT m_Error;
	 UINT w_lMsgLen;

	 USINT m_SendBuffer[300];
	 USINT m_ReadBuffer[300];
	 USINT pb_mBoxDoTextRead[120];
	 BYTE pb_mBoxCont[BUFF_SZ_VS0];
	 WORD w_mBoxSize;
	 WORD w_mBoxCSize;
	 WORD w_mBoxWrite;
	 WORD w_mBoxRead;
	 WORD m_sSize;
     WORD w_lLength;
	 WORD InByteCount_DATA;

	 BYTE m_byType;
	 BYTE m_byRate;
	 BOOL m_blMsgFind;
     STCPADDR m_stTcpAddr;
	 BYTE m_bSrvState;
	 BYTE m_bCliState;
	 SMESSAGE m_sMsg;
	 CMTimer m_nConnTMR;
	 SARMINTERFACE *m_pArm;
	 DECLARE_IMPLEMENT_BASE(CCyclicSystem)
}
DECLARE_DEFINITION(CComVS0)
#endif
```

#### bnrcomvs1.c
```c
/********************************************************************
 * COPYRIGHT -- Kontora
 ********************************************************************
 * Program: bnrmain
 * File: bnrlsens.c
 * Author: Abramenya
 * Created: January 19, 2009
 *******************************************************************/

#include "bnrcomvs1.h"
#ifdef _DEFAULT_INCLUDES
 #include <AsDefault.h>
#endif
extern SINT *chPortType[];
extern SINT *chPortRate[];
extern SINT *chPortParity[];
extern SINT *chPortData[];
extern SINT *chPortStop[];
_GLOBAL FRM_xopen_typ m_sXOpenVS1;
_GLOBAL XOPENCONFIG   m_sConfigVS1;
_GLOBAL FRM_gbuf_typ  m_sFrameBuffVS1;
_GLOBAL FRM_rbuf_typ  m_sRBuffVS1;
_GLOBAL FRM_write_typ m_sSendVS1;
_GLOBAL FRM_read_typ  m_sReccVS1;
_GLOBAL FRM_close_typ m_sCloseVS1;
_GLOBAL FRM_robuf_typ m_sRobuffVS1;
#ifndef WIN32
_GLOBAL FRM_mode_typ FrameModeStructVS1;
#endif

void CComVS1_Init(This,SARMINTERFACE *pArm)
{
    DECLARE_MULTI_OPEN(CComVS1,CCyclicSystem)
    //#ifdef WIN32
	//m_nCommServer = pT;
    //#endif
	pT->m_pArm = pArm;
	FDEFINE(DEV_RSVS1MMD_BOX_ID,1024);
	FDEFINE(DEV_RSVBS1_BOX_ID,1024);
	pB->SetBoxID(pB,DEV_RSVS1MMD_BOX_ID);

	InitObject(CMTimer,&pT->m_nConnTMR);
	pT->m_nConnTMR.SetTimer(&pT->m_nConnTMR,DIR_PHTOPH,DIR_PHTOPH,EV_TMR_SRR_REQ,0,0,DEV_RSVS1MMD_BOX_ID);

	pT->m_blMsgFind = FALSE;
	pT->m_byType = pArm->byType;
	pT->m_byRate = pArm->byPortRate;
	pT->InByteCount_DATA = 0;

	strcpy(pT->m_chStringMode, chPortType[pT->m_pArm->byType]);
	strcat(pT->m_chStringMode,", ");
	strcat(pT->m_chStringMode, chPortRate[pT->m_pArm->byPortRate]);
	strcat(pT->m_chStringMode,", ");
	strcat(pT->m_chStringMode, chPortParity[pT->m_pArm->stTcpAddr.byAddr0]);
	strcat(pT->m_chStringMode,", ");
	strcat(pT->m_chStringMode, chPortData[pT->m_pArm->stTcpAddr.byAddr1]);
	strcat(pT->m_chStringMode,", ");
	strcat(pT->m_chStringMode, chPortStop[pT->m_pArm->stTcpAddr.byAddr2]);

	strcpy(pT->m_chStringDevice, "IF4.ST2");
	#ifdef DEB_CComVS1
	Info("\n(__)CTCPS::>Create %s.Device: %s Mode: %s",
	chPortType[pT->m_byType],pT->m_chStringDevice,pT->m_chStringMode);
	#endif
	pT->SynBuff(pT);
    pT->InitSRV(pT);
	//pT->m_nConnTMR.OnTimer(&pT->m_nConnTMR,200);
	pT->m_StatusWrite = 0;
	pT->m_bSrvState = DRV_ST_CONN;
	pT->m_bCliState = DRV_ST_CONN;
}
void CComVS1_SetPortSett(This)
{
    DECLARE_MULTI_OPEN(CComVS1,CCyclicSystem)
    strcpy(pT->m_chStringDevice, "IF4.ST2");
	memset(pT->m_chStringNewMode,0,sizeof(pT->m_chStringNewMode));

	strcpy(pT->m_chStringNewMode, chPortType[pT->m_pArm->byType]);
	strcat(pT->m_chStringNewMode,", ");
	strcat(pT->m_chStringNewMode, chPortRate[pT->m_pArm->byPortRate]);
	strcat(pT->m_chStringNewMode,", ");
	strcat(pT->m_chStringNewMode, chPortParity[pT->m_pArm->stTcpAddr.byAddr0]);
	strcat(pT->m_chStringNewMode,", ");
	strcat(pT->m_chStringNewMode, chPortData[pT->m_pArm->stTcpAddr.byAddr1]);
	strcat(pT->m_chStringNewMode,", ");
	strcat(pT->m_chStringNewMode, chPortStop[pT->m_pArm->stTcpAddr.byAddr2]);
    #ifndef WIN32
    FrameModeStructVS1.ident  = m_sXOpenVS1.ident;
    FrameModeStructVS1.mode   = (UDINT)pT->m_chStringNewMode;
    FrameModeStructVS1.enable = 1;
    FRM_mode(&FrameModeStructVS1);
    #endif
}
void CComVS1_SynBuff(This)//CANOpen
{
    DECLARE_MULTI_OPEN(CComVS1,CCyclicSystem)
	pT->w_mBoxSize  = BUFF_SZ_VS1;
    pT->w_mBoxCSize = BUFF_SZ_VS1;
	pT->w_mBoxWrite = 0;
	pT->w_mBoxRead  = 0;
	pT->m_sSize     = 0;
	pT->w_lLength   = 0;
	pT->w_lMsgLen   = 0;
	memset(&pT->pb_mBoxCont[0],0,10);
	#ifdef DEB_CComVS1
	Info("\n(__)CTCPS::>Synchro.");
    #endif
}
//_GLOBAL FRM_xopen_typ FrameXOpenStruct;
//_GLOBAL XOPENCONFIG XOpenConfigStruct;
void CComVS1_InitSRV(This)
{
    DECLARE_MULTI_OPEN(CComVS1,CCyclicSystem)
	//Server Init
    m_sConfigVS1.idle     = 10;
    m_sConfigVS1.delimc   = 0;
    m_sConfigVS1.delim[0] = 0;
	m_sConfigVS1.delim[1] = 0;
	m_sConfigVS1.tx_cnt   = 2;
	m_sConfigVS1.rx_cnt   = 2;
	m_sConfigVS1.tx_len   = 256;
	m_sConfigVS1.rx_len   = 256;
	m_sConfigVS1.argc     = 0;
	m_sConfigVS1.argv     = 0;

	strcpy(pT->m_chStringMode, "RS232, 1200, N, 8, 1");
	m_sXOpenVS1.device    = (UDINT) pT->m_chStringDevice;
	m_sXOpenVS1.mode      = (UDINT) pT->m_chStringMode;
    m_sXOpenVS1.config    = (UDINT)&m_sConfigVS1;
	m_sXOpenVS1.enable    = 1;
	pT->m_StatusOpen   = 0;
    #ifndef WIN32
	pT->m_nConnTMR.OnTimer(&pT->m_nConnTMR,30);
    #else
	pT->m_nConnTMR.OnTimer(&pT->m_nConnTMR,30);
	//pT->Open(pT);
    #endif
}
_GLOBAL INT nOPEN,nCLOSE;

BOOL CComVS1_Open(This)
{
    DECLARE_MULTI_OPEN(CComVS1,CCyclicSystem)
	SHORTMESSAGE m_sMsg;
    if(pT->m_StatusOpen==0)
	{
	#ifndef WIN32
	FRM_xopen(&m_sXOpenVS1);
    #endif
	if(m_sXOpenVS1.status==0)
	{
	 nOPEN++;
	 m_sReccVS1.ident      = m_sXOpenVS1.ident;
	 m_sSendVS1.ident      = m_sXOpenVS1.ident;
	 m_sCloseVS1.ident     = m_sXOpenVS1.ident;
	 m_sFrameBuffVS1.ident = m_sXOpenVS1.ident;
	 m_sRBuffVS1.ident     = m_sXOpenVS1.ident;
	 m_sReccVS1.buffer	    = (UDINT)&pT->m_ReadBuffer[0];
	 m_sSendVS1.buffer     = (UDINT)&pT->m_SendBuffer[0];
	 m_sFrameBuffVS1.buffer= m_sSendVS1.buffer;
	 m_sRBuffVS1.buffer    = m_sReccVS1.buffer;
	 m_sReccVS1.enable     = 1;
	 m_sSendVS1.enable     = 1;
	 m_sCloseVS1.enable    = 1;
	 m_sFrameBuffVS1.enable= 1;
	 m_sRBuffVS1.enable    = 1;
	 pT->m_StatusOpen   = 1;
	 pT->m_StatusWrite  = 0;
	 //pT->SendSMessage(pT,DEV_KPMDL_BOX_ID,DIR_PHTOKP,PH_CALL_REQ);
	 return TRUE;
	}
 	}
	return FALSE;
}
void CComVS1_Enable(This)
{
	DECLARE_MULTI_OPEN(CComVS1,CCyclicSystem)
	m_sXOpenVS1.enable = 1;
}
void CComVS1_Disable(This)
{
	DECLARE_MULTI_OPEN(CComVS1,CCyclicSystem)
	m_sXOpenVS1.enable = 0;
}
void CComVS1_Close(This)
{
    DECLARE_MULTI_OPEN(CComVS1,CCyclicSystem)
	m_sCloseVS1.enable = 1;
	FRM_close(&m_sCloseVS1);
}
BOOL CComVS1_SendMessage(This,SMESSAGE *pMsg)
{
	DECLARE_MULTI_OPEN(CComVS1,CCyclicSystem)
	BOOL res = TRUE;
	if(pT->m_StatusOpen==1)
	{
	 FRM_gbuf(&m_sFrameBuffVS1);
     m_sSendVS1.buflng = pMsg->m_swLen-9;
	 memcpy(m_sSendVS1.buffer, &pMsg->m_sbyInfo[0],m_sSendVS1.buflng);
	 FRM_write(&m_sSendVS1);
	 pT->m_StatusWrite  = m_sSendVS1.status;
	 if(pT->m_StatusWrite==0) res = TRUE;else res = FALSE;
	}
	return res;
}
_GLOBAL INT nSNDVS0;
_GLOBAL INT nSendThreadVS0;
void CComVS1_SendThread(This)
{
    DECLARE_MULTI_OPEN(CComVS1,CCyclicSystem)
	nSendThreadVS0++;
    //if(pT->m_StatusWrite==0)
	if(pT->m_StatusOpen==1)
    {
	 if(FGET(DEV_RSBUF_BOX_ID,&pT->m_sMsg))
	 {
	  //Info("\n(__)CRSVO::>TX:%M",&pT->m_sMsg);
	  if(pT->m_sMsg.m_swLen<=256)
	  {
	   nSNDVS0++;
       pT->SendMessage(pT,&pT->m_sMsg);
	  }//else
	    //Info("\n(__)CRSVO::>Wery Long Message!");
	 }
	}
 	 //else
 	 //{
 	 // #ifdef DEB_CComVS1
 	 // ///Info("\n(__)Wait.");
 	 // #endif
 	 //}
}
_GLOBAL INT nGETL1VS0;
BOOL CComVS1_GetMessage(This,SMESSAGE *pMsg)
{
    DECLARE_MULTI_OPEN(CComVS1,CCyclicSystem)
	BYTE i,*pBuff;
	BOOL res=FALSE;
	SMESSAGE csM;
	if(pT->m_StatusOpen==1)
	{
	FRM_read(&m_sReccVS1);
	pT->m_StatusRead       = m_sReccVS1.status;
	if(pT->m_StatusRead==0)
	{
	 pT->m_ReadBufferLength = m_sReccVS1.buflng;
	 pBuff                  = m_sReccVS1.buffer;
	 /*
	 csM.m_sbyInfo[0] = 0x7e;
	 csM.m_sbyInfo[1] = 'A';
	 csM.m_sbyInfo[2] = 'l';
	 csM.m_sbyInfo[3] = 'e';
	 csM.m_sbyInfo[4] = 'x';
	 csM.m_sbyInfo[5] = 'a';
	 csM.m_sbyInfo[6] = 'n';
	 csM.m_sbyInfo[7] = 'd';
	 csM.m_sbyInfo[8] = 'e';
	 csM.m_sbyInfo[9] = 'r';
	 csM.m_sbyInfo[10] = 0xe7;
	 */

	 //memcpy(&csM.m_sbyInfo[0],m_sReccVS1.buffer,pT->m_ReadBufferLength);
	 //csM.m_swLen = 9 + pT->m_ReadBufferLength;
	 //Info("\n(__)CRSVO::>MSG:%M",&csM);

	 //m_sRBuffVS1.buffer = m_sReccVS1.buffer;
	 //m_sRBuffVS1.buflng = pT->m_ReadBufferLength;
	 //FRM_rbuf(&m_sRBuffVS1);
	 //res = TRUE;
	 //nGETL1++;
	 //Info("\nMSG::>");
	 //csM.m_swLen = pT->m_ReadBufferLength+9;
	 for( i=0;i<pT->m_ReadBufferLength;i++)
	 {
	  pT->pb_mBoxCont[pT->w_mBoxWrite] = pBuff[i];
      //Info(" %b",&pT->pb_mBoxCont[pT->w_mBoxWrite]);
	  //printf(" %c",pT->pb_mBoxCont[pT->w_mBoxWrite]);
      pT->w_mBoxWrite = (pT->w_mBoxWrite + 1) & BUFF_SZ_VS1;
	 }
	 //FPUT(DEV_RSBUF_BOX_ID,(BYTE*)&csM);
	 pT->w_mBoxSize -= pT->m_ReadBufferLength;
	 pT->m_sSize     = pT->w_mBoxCSize-pT->w_mBoxSize;
	 //Info("\nRD::>%b PRD::>%w PWD::>%w FND::>%b",&pT->pb_mBoxCont[pT->w_mBoxRead],&pT->w_mBoxRead,&pT->w_mBoxWrite,&pT->m_blMsgFind);
	 if ((pT->pb_mBoxCont[pT->w_mBoxRead]==0x3d))
	 {
		 pT->m_blMsgFind = TRUE;
		 if(res = pT->MakeMsgData(pT,pMsg))
		 {
			 pT->m_blMsgFind = FALSE;
			 res = TRUE;
		 }
	 }else
		 pT->SynBuff(pT);
	 m_sRBuffVS1.buffer = m_sReccVS1.buffer;
	 m_sRBuffVS1.buflng = pT->m_ReadBufferLength;
	 FRM_rbuf(&m_sRBuffVS1);
     }
	}
	return res;
}
BOOL CComVS1_MakeMsgData(This,SMESSAGE *pMsg)
{
    DECLARE_MULTI_OPEN(CComVS1,CCyclicSystem)
	WORD lLen,i,nCM=0;
	BOOL res = FALSE;
	lLen = 1;
	pT->w_lMsgLen = pT->w_lMsgLen + pT->m_ReadBufferLength;
	if (pT->w_lMsgLen>BUFF_SZ_VS1) {pT->SynBuff(pT);return res;}
    for (i=1;i<pT->w_lMsgLen-1;i++)
	{
	 lLen++;
	 if (pT->pb_mBoxCont[(pT->w_mBoxRead+i)& BUFF_SZ_VS1]==0x2e) nCM++;
	 if (nCM>1){pT->SynBuff(pT);return res;}
	 if (lLen>300) {pT->SynBuff(pT);return res;}
     if (pT->pb_mBoxCont[(pT->w_mBoxRead+i)& BUFF_SZ_VS1]==0x3d)
     {
	  pT->CopyMessage(pT,lLen,pMsg);
	  //pT->SynBuff(pT);
	  pT->w_lMsgLen = 0;
	  return TRUE;
	 }
	}
	return res;
}
BOOL CComVS1_CopyMessage(This,WORD wLen,SMESSAGE *pMsg)
{
    DECLARE_MULTI_OPEN(CComVS1,CCyclicSystem)
	INT i,j=0;BYTE byCRC;
	BOOL blCRC;
	for(i=0;i<wLen;i++)
	{
		if ((i!=0)&&(i!=wLen-1)){pMsg->m_sbyInfo[j]=pT->pb_mBoxCont[pT->w_mBoxRead];j++;}
		pT->w_mBoxSize =(pT->w_mBoxSize+1)& BUFF_SZ_VS1;
		pT->w_mBoxRead=(pT->w_mBoxRead+1)& BUFF_SZ_VS1;
		//Info(" %b",&pMsg->m_sbyInfo[i]);
		//printf(" %x",pMsg->m_sbyInfo[i]);
	}
	pMsg->m_sbyInfo[j++] = 0x00;
	pT->w_mBoxRead=(pT->w_mBoxRead-1)& BUFF_SZ_VS1;
	pT->m_sSize = (pT->w_mBoxCSize-pT->w_mBoxSize) & BUFF_SZ_VS1;
	pMsg->m_swLen         = j+9;
	pMsg->m_sbyFrom       = DIR_PHMDL;
	pMsg->m_sbyFor        = DIR_PHTOMS;
	pMsg->m_sbyIntType    = 0;
	pMsg->m_sbyServerID   = 0;
	pMsg->m_sbyType       = PH_VS1_REQ;
	pMsg->m_sbyDirection  = 0;
	pMsg->m_sbySensor     = 0;
	return TRUE;
}
BYTE CComVS1_CreateCRC(This,BYTE *pMsg,BYTE byLen)
{
	DECLARE_MULTI_OPEN(CComVS1,CCyclicSystem)
	BYTE i,sum = 0;
	for(i=0;i<=byLen-1;i++)sum += pMsg[i];
	return sum;
}
_GLOBAL INT nReceiveThreadVS0;
void CComVS1_ReceiveThread(This)
{
    DECLARE_MULTI_OPEN(CComVS1,CCyclicSystem)
	nReceiveThreadVS0++;
	#ifndef WIN32
	if(pT->GetMessage(pT,&pT->m_sMsg)==TRUE)
	{
	 //Info("\n(__)CRSVO::>RX:%M",&pT->m_sMsg);
	 FPUT(DEV_MSMDL_BOX_ID,(BYTE*)&pT->m_sMsg);
		//FPUT(DEV_RSBUF_BOX_ID,(BYTE*)&pT->m_sMsg);
	}
    #endif
}
_GLOBAL INT nRSEventHandlerVS0,nCheckOpenVS0,nWatchOpenVS0;
BOOL CComVS1_EventHandler(This,SMESSAGE *pMsg)
{
    DECLARE_MULTI_OPEN(CComVS1,CCyclicSystem)
	switch(pMsg->m_sbyFor)
	{
	  case DIR_101TOPH:
	       #ifdef DEB_CComVS1
		   Info("\n(__)CRSVO::>OUTP::%M",pMsg);
		   #endif
		   FPUT(DEV_RSBUF_BOX_ID,pMsg);
	  break;
	  case DIR_PHTOPH:
	       if (pMsg->m_sbyType==EV_TMR_SRR_REQ)
		   {
		   	//if(pT->m_StatusOpen==0)
			{
			 nCheckOpenVS0++;
 		     pT->Open(pT);
			}
			pT->m_nConnTMR.OnTimer(&pT->m_nConnTMR,30);
		   }
	  break;
      case DIR_KPTOPH:
	       if (pMsg->m_sbyType==PH_CLOSE_PORT_REQ)
		   {
            //pT->Close(pT);
		   }
		   if(pMsg->m_sbyType==PH_INIT_PORT_REQ)
		   {
             pT->SetPortSett(pT);
		   }
	  break;
	  default:
	  break;
	}
	return TRUE;
}
void CComVS1_Connect(This)
{
    DECLARE_MULTI_OPEN(CComVS1,CCyclicSystem)
    SHORTMESSAGE m_sMsg;
	m_sMsg.m_swLen        = 9;
	m_sMsg.m_sbyFrom      = DIR_PHMDL;
	m_sMsg.m_sbyFor       = DIR_PHTO101P;
	m_sMsg.m_sbyIntType   = 0;
	m_sMsg.m_sbyServerID  = 0;
	m_sMsg.m_sbyType      = PH_CONN_IND;
	m_sMsg.m_sbyDirection = 0;
	m_sMsg.m_sbySensor    = 0;
	FPUT(DEV_101MD_BOX_ID,(BYTE*)&m_sMsg);
    #ifdef DEB_CComVS1
	Info("\n(__)CRSVO::>OUTT::%M",&m_sMsg);
    #endif
}
void CComVS1_SendSMessage(This,BYTE byBox,BYTE byFor,BYTE byType)
{
    DECLARE_MULTI_OPEN(CComVS1,CCyclicSystem)
    SHORTMESSAGE m_sMsg;
	m_sMsg.m_swLen        = 9;
	m_sMsg.m_sbyFrom      = DIR_PHMDL;
	m_sMsg.m_sbyFor       = byFor;
	m_sMsg.m_sbyIntType   = 0;
	m_sMsg.m_sbyServerID  = 0;
	m_sMsg.m_sbyType      = byType;
	m_sMsg.m_sbyDirection = 0;
	m_sMsg.m_sbySensor    = 0;
	FPUT(byBox,(BYTE*)&m_sMsg);
    #ifdef DEB_CComVS1
	Info("\n(__)CRSVO::>OUTT::%M",&m_sMsg);
    #endif
}
void CComVS1_Disconnect(This)
{
    DECLARE_MULTI_OPEN(CComVS1,CCyclicSystem)
    SHORTMESSAGE m_sMsg;
	m_sMsg.m_swLen        = 9;
	m_sMsg.m_sbyFrom      = DIR_PHMDL;
	m_sMsg.m_sbyFor       = DIR_PHTO101P;
	m_sMsg.m_sbyIntType   = 0;
	m_sMsg.m_sbyServerID  = 0;
	m_sMsg.m_sbyType      = PH_DISC_IND;
	m_sMsg.m_sbyDirection = 0;
	m_sMsg.m_sbySensor    = 0;
	FPUT(DEV_101MD_BOX_ID,(BYTE*)&m_sMsg);
    #ifdef DEB_CComVS1
	Info("\n(__)CRSVO::>OUTT::%M",&m_sMsg);
    #endif
}
void CComVS1_CyclicProc(This)
{
    DECLARE_MULTI_OPEN(CComVS1,CCyclicSystem)
	pT->ReceiveThread(pT);
}
void CComVS1_CComVS1(This)
{
    DECLARE_MULTI_OPEN(CComVS1,CCyclicSystem)
	DECLARE_REGISTRATION(CComVS1,Init)
	DECLARE_REGISTRATION(CComVS1,InitSRV)
	DECLARE_REGISTRATION(CComVS1,SendMessage)
	DECLARE_REGISTRATION(CComVS1,GetMessage)
    DECLARE_REGISTRATION(CComVS1,Close)
	DECLARE_REGISTRATION(CComVS1,Disable)
	DECLARE_REGISTRATION(CComVS1,Enable)
	DECLARE_REGISTRATION(CComVS1,Open)
	DECLARE_REGISTRATION(CComVS1,ReceiveThread)
	DECLARE_REGISTRATION(CComVS1,SendThread)
	DECLARE_REGISTRATION(CComVS1,SynBuff)
	DECLARE_REGISTRATION(CComVS1,MakeMsgData)
	DECLARE_REGISTRATION(CComVS1,CopyMessage)
	DECLARE_REGISTRATION(CComVS1,CreateCRC)
	DECLARE_REGISTRATION(CComVS1,Connect)
	DECLARE_REGISTRATION(CComVS1,Disconnect)
	DECLARE_REGISTRATION(CComVS1,SendSMessage)
	DECLARE_REGISTRATION(CComVS1,SetPortSett)
	DECLARE_VIRTUAL_FUNC(CComVS1,EventHandler)
	DECLARE_VIRTUAL_FUNC(CComVS1,CyclicProc)
}

void CComVS1_DCComVS1(This)
{
	DECLARE_MULTI_OPEN(CComVS1,CCyclicSystem)
	//DESTROY
}

DECLARE_MULTI_CREATE(CComVS1,CCyclicSystem)
```

#### bnrdevtu.h
```c
/********************************************************************
 * COPYRIGHT -- Kontora
 ********************************************************************
 * Program: bnrmain
 * File: bnraninput.h
 * Author: Abramenya
 * Created: January 19, 2009
 *******************************************************************/

#ifndef __DEVTU_H__
#define __DEVTU_H__
#include "typedefs.h"
#include "bnrtelesensor.h"
/*
enum _enTUCommand
{
     EN_STT_PULCE=9,
	 EN_STT_SIGN =10,
};
*/
#define DEF_PULCE 20
/*
//Телеуправление1(дискретное)
typedef struct _tagTUMData
{
	BYTE byParam;
}STUMDATA;
typedef struct _tagTUMParam
{
	BYTE byID;
	BYTE byAmParam;
	BYTE byType;
	BYTE bySlot;
	BYTE byPin;
	BYTE byAlmState;
	BYTE byState;
	BYTE byPulceType;
    BYTE byCSetPulce;
	STUMDATA sDT;
}STUMPARAM;
*/
Class CDevTU
{
	 void (*CCDevTU)(This);
	 void (*DCDevTU)(This);
Public
     void (*Init)(This,BOOL *pblValue,BYTE byID,BYTE byIID,BYTE byState,BYTE byPulceType,DWORD byCSetPulce);
	 void (*SetTU)(This,BYTE byBox,BYTE byFor,BYTE byEv);
     void (*PreProc)(This);
     void (*Processing)(This);
	 void (*PostProc)(This);
	 void (*SendEvent)(This,SKPEVENT *pEV);
	 BOOL (*SaveChange)(This,BYTE byEvent,WORD wValue,BOOL blAlarm);
     void (*SetPulce)(This);
     void (*PreparePulce)(This);
     void (*SetPulceEx)(This,DWORD wPulce);
     void (*SetPin)(This);
     void (*InvPin)(This);
	 DWORD (*Run)(This);
	 void (*Stop)(This);
Public
	 STUMPARAM pP;
     BYTE m_byBox;
	 BYTE m_byFor;
	 BYTE m_byEv;
	 BYTE m_byID;
	 BYTE m_byPinID;
     BYTE m_byOldEvent;
     DWORD m_bySetPulce;
	 DWORD m_dwJob;
	 BYTE m_byStPulce;
	 BYTE m_byType;
	 BOOL *m_pbOT;
	 DECLARE_IMPLEMENT
	 //DECLARE_IMPLEMENT_BASE(CTeleSensor)
}
DECLARE_DEFINITION(CDevTU)
#endif
```
